//Error
IF timDissableFunctions.Q THEN 
	fbBattery.bWarning := TRUE; 
	fbBattery.iWarningCode := 0; 
ELSE 
	fbBattery.bWarning := FALSE; 
END_IF 
IF (stDataPixii.bError AND stDataPixii.eBatteryState = E_Pixii_BatteryState.eFault) OR timErrorMTCP.Q OR Lynus_Standards.GVL_Energy.stNumberOfDevices.diNumberOfBatterys > Constants_Energy.diMaxNumberOfBatterys THEN 
	fbBattery.bError := TRUE; 
ELSE 
	fbBattery.bError := FALSE; 
END_IF
IF Lynus_Standards.GVL_Energy.stNumberOfDevices.diNumberOfBatterys > Constants_Energy.diMaxNumberOfBatterys THEN 
	fbBattery.iErrorCode := 1;
ELSIF stDataPixii.bError THEN 
	fbBattery.iErrorCode := 0; 
END_IF

//Function
fbBattery(
	bEnable:= bEnable AND NOT timDissableFunctions.Q, 
	bError:= , 
	bWarning:= , 
	bCalculatePower:= TRUE, 
	bReset:= bReset OR timReset.Q, 
	bWriteWithDelay:= TRUE, 
	iErrorCode:= , 
	iWarningCode:= , 
	dwBatterySOC:= , 
	dwBatterySOH:= 0, 
	rBatteryVoltage:= , 
	rMaxDcChargeCurrentBattery:= , 
	rMaxDcDischargeCurrentBattery:= , 
	rMaxChargeVoltage:= 0, 
	lrMaxCapacityBattery:= lrMaxCapacityBattery, 
	lrBatteryPower:= 0, 
	lrBatteryCurrent:= , 
	lrBatteryTemp:= , 
	tTimDelayOutput:= T#5S, 
	stDataBatteryOut=> , 
	stDataBatteryOutDelay=> stDataBatt);


(*------------------------------------------------------------------------------------------State Machine Write---------------------------------------------------------------------------------------------*)	
	
CASE iStateModbusWrite OF	
	
	1://Setpoint for Power 
		iStateModbus_CP := iStateModbusWrite;	
		
		//fbMBWrite_FC6.nQuantity := 2;
		fbMBWrite_FC6.nMBAddr := 39904;
		fbMBWrite_FC6.bExecute := TRUE;
	
		//Setpoint for the Power when discharge (in kW on the Inverter) 
		IF fbBatteryInverter.stDataBattInvertOut.rTargetPower >= 0 THEN
			IF 	((fbBatteryInverter.stDataBattInvertOut.rMaxDischargePower /100) * (fbBatteryInverter.stDataBattInvertOut.rTargetPower * 100)) >= - 32768 AND 
				((fbBatteryInverter.stDataBattInvertOut.rMaxDischargePower /100) * (fbBatteryInverter.stDataBattInvertOut.rTargetPower * 100)) <= 32767 THEN
					iSetpointPower := REAL_TO_INT((fbBatteryInverter.stDataBattInvertOut.rMaxDischargePower / 100) * (fbBatteryInverter.stDataBattInvertOut.rTargetPower * 100));  
					wordBuffer_FC6 := INT_TO_WORD(iSetpointPower);
			END_IF
		END_IF
		//Setpoint for the Power when charge (in kW on the Inverter) 
		IF fbBatteryInverter.stDataBattInvertOut.rTargetPower < 0 OR fbPIDChrgStandby.bEnable THEN
			IF 	((fbBatteryInverter.stDataBattInvertOut.rMaxChargePower / 100) * (fbBatteryInverter.stDataBattInvertOut.rTargetPower * 100)) >= - 32768 AND 
				((fbBatteryInverter.stDataBattInvertOut.rMaxChargePower / 100) * (fbBatteryInverter.stDataBattInvertOut.rTargetPower * 100)) <= 32767 THEN
					iSetpointPower := REAL_TO_INT((fbBatteryInverter.stDataBattInvertOut.rMaxChargePower / 100) * (fbBatteryInverter.stDataBattInvertOut.rTargetPower * 100));  
					//Take the Setpoint from the Standby Controller
					IF fbPIDChrgStandby.bEnable AND fbPIDChrgStandby.rQController <= 0 AND fbPIDChrgStandby.rQController >= -32768 THEN
						iSetpointPower := REAL_TO_INT(fbPIDChrgStandby.rQController);  
					END_IF
					wordBuffer_FC6 := INT_TO_WORD(iSetpointPower); 
			END_IF
		END_IF
		//manual operation setpoint, for testing pupose only!
		IF m_ManualSetpointEnable THEN
			wordBuffer_FC6 := INT_TO_WORD(i_SetpointPower_Manual_kW*10); 
		END_IF
		iSetpointPower_Info := WORD_TO_INT(WordBuffer_FC6);
		
		IF fbMBWrite_FC6.bBusy THEN 
			timDelay.IN := TRUE; 
		END_IF

		//Wait for Delay and then next step
		IF NOT fbMBWrite_FC6.bBusy AND NOT fbMBWrite_FC6.bError AND timDelay.Q THEN
			fbMBWrite_FC6.bExecute := FALSE;
			timDelay.IN := FALSE;
			stDataPixii.bError := FALSE; 
			stDataPixii.eErrorState := E_Pixii_Error.eNormal;
			//Restart from new with the Read out part
			iStateModbusRead := 0;
			iStateModbusWrite := 10;
		END_IF
				
		//Error or Timout
		IF FPError_FC_6.Q OR timTimeout.Q THEN
			iStateModbusError := 300;
			stDataPixii.eErrorState := E_Pixii_Error.eModbusTCPError;
		END_IF

	10:// waite one cycle and count handshake counter +1
		int_Handshake_Counter := int_Handshake_Counter+1;
		iStateModbusWrite := 11;
	
	11:// write handshake timeout +1
		iStateModbus_CP := iStateModbusWrite;	
		
		//fbMBWrite_FC6.nQuantity := 2;
		fbMBWrite_FC6.nMBAddr := 39903;
		fbMBWrite_FC6.bExecute := TRUE;
	
		wordBuffer_FC6 := INT_TO_WORD(int_Handshake_Counter); 
		
		IF fbMBWrite_FC6.bBusy THEN 
			timDelay.IN := TRUE; 
		END_IF

		//Wait for Delay and then next step
		IF NOT fbMBWrite_FC6.bBusy AND NOT fbMBWrite_FC6.bError AND timDelay.Q THEN
			fbMBWrite_FC6.bExecute := FALSE;
			timDelay.IN := FALSE;
			stDataPixii.bError := FALSE; 
			stDataPixii.eErrorState := E_Pixii_Error.eNormal;
			//Restart from new with the Read out part
			iStateModbusRead := 1;
			iStateModbusWrite := 0;
		END_IF
				
		//Error or Timout
		IF FPError_FC_6.Q OR timTimeout.Q THEN
			iStateModbusError := 300;
			stDataPixii.eErrorState := E_Pixii_Error.eModbusTCPError;
		END_IF

END_CASE

(*------------------------------------------------------------------------------------------State Machine Write---------------------------------------------------------------------------------------------*)	

CASE iStateModbusError OF
	
	300://Error
		iStateModbus_CP := iStateModbusError;
		timDelay.IN := FALSE;
		fbMBRead_FC3.bExecute := FALSE;
		fbMBWrite_FC6.bExecute := FALSE;
		stDataPixii.bError := TRUE;	
		//Restart from new with the Read out part after an Error
		iStateModbusRead := 1;	
		iStateModbusError := 0;
		iStateModbusWrite := 0;
END_CASE

(*------------------------------------------------------------------------------------------Modbus TCP Functions---------------------------------------------------------------------------------------------*)

fbMBRead_FC3(	sIPAddr:= sIPAdress, 
				nUnitID := byUnitID, 
				nTCPPort:= 502, 
				cbLength:= SIZEOF(arrBuffer_FC3), 
				pDestAddr:= ADR(arrBuffer_FC3), 
				tTimeout:= T#10S );
FPError_FC_3(	CLK:= fbMBRead_FC3.bError, 
				Q=> );

fbMBWrite_FC6(	sIPAddr:= sIPAdress, 
				nTCPPort:= 502, 
				nUnitID:= byUnitID, 
				nMBAddr:= , 
				nValue:= wordBuffer_FC6, 
				bExecute:= , 
				tTimeout:=  T#10S, 
				bBusy=> , 
				bError=> , 
				nErrId=> );				

FPError_FC_6(	CLK:= fbMBWrite_FC6.bError, 
				Q=> );


				
//Function
fbEMPower(
	bEnable:= bEnable AND NOT timDissableFunctions.Q, 
	bError:= , 
	bEnableReadOutFunction:= FALSE, 
	bWriteWithDelay:= TRUE, 
	bPowerDataInvers:= FALSE,
	bReadOutDataDone:= ,
	iTimeReadOutInterval:= , 
	iErrorCode:= , 
	iWarningCode:= , 
	lrTotalCounterEnergy_Consumption:= , 
	lrTotalCounterEnergy_Production:= , 
	lrCounterEnergyT1_Consumption:= , 
	lrCounterEnergyT2_Consumption:= 0, 
	lrCounterEnergyT1_Production:= , 
	lrCounterEnergyT2_Production:= 0, 
	lrCurrentL1:= , 
	lrVoltageL1N:= , 
	lrVoltageL1L2:= , 
	lrPowerL1:= 0, 
	lrCurrentL2:= , 
	lrVoltageL2N:= , 
	lrVoltageL2L3:= , 
	lrPowerL2:= 0, 
	lrCurrentL3:= , 
	lrVoltageL3N:= , 
	lrVoltageL3L1:= , 
	lrPowerL3:= 0, 
	lrPowerTotal:= , 
	lrFrequency:= , 
	lrReactivePowerTotal:= , 
	lrApparentPowerTotal:= 0, 
	tTimDelayOutput:= T#5S, 
	stDataEMOutPower=> , 
	stDataEMOutPowerDelay=> stDataEMPower, 
	stDataEMOutCounter=> ,
	stDataEMOutCounterDelay=> stDataEMCounter,  
	bReadOutMeter=> );
(*-----------------------------------------------------------Handle data to Global structure for al Devices that are included in this function-----------------------------------------------------------------*)

//Delete al old Data on GVL after a online change or change on the variable diNrOfEMS_IDOD
IF diNrOfEMS_IN <> diNrOfEMS_IN_CP AND iStateGVLData = 0 THEN 
	iStateGVLData := 10; 
END_IF 

CASE iStateGVLData OF
	
	0://Init Step
		byWaitInStep := 0;
		arrCounterForGVL[1] := 1; arrCounterForGVL[2] := 1; arrCounterForGVL[3] := 1;
	
	1://Wait for 4 Steps before clean al Data on GVL
		byWaitInStep := byWaitInStep + 1;
		IF (byWaitInStep >= 4 AND (fbNumberDeviceBattery.bNumberIsCalculatet OR fbNumberDeviceBatteryInvert.bNumberIsCalculatet OR fbNumberDeviceGrid.bNumberIsCalculatet)) THEN 
			iStateGVLData := 2; 
		END_IF
		//To much Devices, back to the Init step
		IF byWaitInStep >= 4 AND NOT fbNumberDeviceBattery.bNumberIsCalculatet AND NOT fbNumberDeviceBatteryInvert.bNumberIsCalculatet AND NOT fbNumberDeviceGrid.bNumberIsCalculatet THEN 
			iStateGVLData := 0; 
		END_IF	
			
	2://Clear all Data in GVL
		FOR diLPForGVL := 1 TO Constants_Energy.diMaxNumberOfEMS BY 1 DO
			//Battery Inverters 
			IF fbNumberDeviceBatteryInvert.bNumberIsCalculatet THEN 
				Lynus_Standards.GVL_Energy.stDataOfBatteryInverters[diLPForGVL,arrCounterForGVL[1]].bEnabled := FALSE;
				Lynus_Standards.GVL_Energy.stDataOfBatteryInverters[diLPForGVL,arrCounterForGVL[1]].bOnOff := FALSE;
				Lynus_Standards.GVL_Energy.stDataOfBatteryInverters[diLPForGVL,arrCounterForGVL[1]].bWorkOnIslandMode := FALSE;
				Lynus_Standards.GVL_Energy.stDataOfBatteryInverters[diLPForGVL,arrCounterForGVL[1]].byErrorWarning := 0;
				Lynus_Standards.GVL_Energy.stDataOfBatteryInverters[diLPForGVL,arrCounterForGVL[1]].byPriority := 0;
				Lynus_Standards.GVL_Energy.stDataOfBatteryInverters[diLPForGVL,arrCounterForGVL[1]].dwBatterySOC := 0;
				Lynus_Standards.GVL_Energy.stDataOfBatteryInverters[diLPForGVL,arrCounterForGVL[1]].lrPowerOnIslandMode := 0;
				Lynus_Standards.GVL_Energy.stDataOfBatteryInverters[diLPForGVL,arrCounterForGVL[1]].rMaxChargePower := 0;
				Lynus_Standards.GVL_Energy.stDataOfBatteryInverters[diLPForGVL,arrCounterForGVL[1]].rMaxDischargePower := 0;
				Lynus_Standards.GVL_Energy.stDataOfBatteryInverters[diLPForGVL,arrCounterForGVL[1]].lrPowerNormalMode := 0;
				//Set also the target value from ems back here to 0 and not in EMS function because EMS is in Standy when we have a online change (Problem when we delete a ems function and make a online change)
				Lynus_Standards.GVL_Energy.stDataOfBatteryInverters[diLPForGVL,arrCounterForGVL[1]].rTargetPowerEMS := 0;
				Lynus_Standards.GVL_Energy.stDataOfBatteryInverters[diLPForGVL,arrCounterForGVL[1]].byMaxDepthOfDischargeEPO := 0;
				Lynus_Standards.GVL_Energy.stDataOfBatteryInverters[diLPForGVL,arrCounterForGVL[1]].byReserveSOCEPO := 0;
			END_IF
			//Batterys 
			IF fbNumberDeviceBattery.bNumberIsCalculatet THEN 
				Lynus_Standards.GVL_Energy.stDataOfBatterys[diLPForGVL,arrCounterForGVL[2]].bEnabled := FALSE;
				Lynus_Standards.GVL_Energy.stDataOfBatterys[diLPForGVL,arrCounterForGVL[2]].byErrorWarning := 0;
				Lynus_Standards.GVL_Energy.stDataOfBatterys[diLPForGVL,arrCounterForGVL[2]].dwSOC := 0;
				Lynus_Standards.GVL_Energy.stDataOfBatterys[diLPForGVL,arrCounterForGVL[2]].dwSOH := 0;
				Lynus_Standards.GVL_Energy.stDataOfBatterys[diLPForGVL,arrCounterForGVL[2]].lrCapacity := 0;
				Lynus_Standards.GVL_Energy.stDataOfBatterys[diLPForGVL,arrCounterForGVL[2]].lrCurrent := 0;
				Lynus_Standards.GVL_Energy.stDataOfBatterys[diLPForGVL,arrCounterForGVL[2]].lrPower := 0;
				Lynus_Standards.GVL_Energy.stDataOfBatterys[diLPForGVL,arrCounterForGVL[2]].lrPowerConsumption := 0;
				Lynus_Standards.GVL_Energy.stDataOfBatterys[diLPForGVL,arrCounterForGVL[2]].lrPowerProduction := 0;
				Lynus_Standards.GVL_Energy.stDataOfBatterys[diLPForGVL,arrCounterForGVL[2]].lrTemp := 0;
				Lynus_Standards.GVL_Energy.stDataOfBatterys[diLPForGVL,arrCounterForGVL[2]].rMaxChargeVoltage := 0;
				Lynus_Standards.GVL_Energy.stDataOfBatterys[diLPForGVL,arrCounterForGVL[2]].rMaxDcChargeCurrent := 0;
				Lynus_Standards.GVL_Energy.stDataOfBatterys[diLPForGVL,arrCounterForGVL[2]].rMaxDcDischargeCurrent := 0;
				Lynus_Standards.GVL_Energy.stDataOfBatterys[diLPForGVL,arrCounterForGVL[2]].rVoltage := 0;
			END_IF
		END_FOR
		//Electric Meter Grid
		IF fbNumberDeviceGrid.bNumberIsCalculatet THEN 
			Lynus_Standards.GVL_Energy.stDataElectricMeters[arrCounterForGVL[3]].bEnabled := FALSE;	
			Lynus_Standards.GVL_Energy.stDataElectricMeters[arrCounterForGVL[3]].byErrorWarning := 0;
			Lynus_Standards.GVL_Energy.stDataElectricMeters[arrCounterForGVL[3]].lrCounterEnergyT1_Consumption := 0;
			Lynus_Standards.GVL_Energy.stDataElectricMeters[arrCounterForGVL[3]].lrCounterEnergyT1_Production := 0;
			Lynus_Standards.GVL_Energy.stDataElectricMeters[arrCounterForGVL[3]].lrCounterEnergyT2_Consumption := 0;
			Lynus_Standards.GVL_Energy.stDataElectricMeters[arrCounterForGVL[3]].lrCounterEnergyT2_Production := 0;
			Lynus_Standards.GVL_Energy.stDataElectricMeters[arrCounterForGVL[3]].lrPower := 0;
			Lynus_Standards.GVL_Energy.stDataElectricMeters[arrCounterForGVL[3]].lrPowerConsumption := 0;
			Lynus_Standards.GVL_Energy.stDataElectricMeters[arrCounterForGVL[3]].lrPowerProduction := 0;
			Lynus_Standards.GVL_Energy.stDataElectricMeters[arrCounterForGVL[3]].lrTotalCounterEnergy_Consumption := 0;
			Lynus_Standards.GVL_Energy.stDataElectricMeters[arrCounterForGVL[3]].lrTotalCounterEnergy_Production := 0;
		END_IF
		
		//Counter for Battery Inverter
		arrCounterForGVL[1] := arrCounterForGVL[1] + 1;
		arrCounterForGVL[1] := LIMIT(0,arrCounterForGVL[1],Constants_Energy.diMaxNumberOfBatteryInverters);
		//Counter for Batterys
		arrCounterForGVL[2] := arrCounterForGVL[2] + 1;
		arrCounterForGVL[2] := LIMIT(0,arrCounterForGVL[2],Constants_Energy.diMaxNumberOfBatterys);
		//Electric Meters
		arrCounterForGVL[3] := arrCounterForGVL[3] + 1;
		arrCounterForGVL[3] := LIMIT(0,arrCounterForGVL[3],Constants_Energy.diMaxNumberOfElectricMeters);
		//Back to the init step
		IF arrCounterForGVL[1] >= Constants_Energy.diMaxNumberOfBatteryInverters AND arrCounterForGVL[2] >= Constants_Energy.diMaxNumberOfBatterys AND arrCounterForGVL[3] >= Constants_Energy.diMaxNumberOfElectricMeters THEN 
			iStateGVLData := 0; 
		END_IF

	10://Clear old Data on GVL 		
		//Battery Inverter
		Lynus_Standards.GVL_Energy.stDataOfBatteryInverters[diNrOfEMS_IN_CP,diNrOfBattInverter_OUT].bEnabled := FALSE;
		Lynus_Standards.GVL_Energy.stDataOfBatteryInverters[diNrOfEMS_IN_CP,diNrOfBattInverter_OUT].bOnOff := FALSE;
		Lynus_Standards.GVL_Energy.stDataOfBatteryInverters[diNrOfEMS_IN_CP,diNrOfBattInverter_OUT].bWorkOnIslandMode := FALSE;
		Lynus_Standards.GVL_Energy.stDataOfBatteryInverters[diNrOfEMS_IN_CP,diNrOfBattInverter_OUT].byErrorWarning := 0;
		Lynus_Standards.GVL_Energy.stDataOfBatteryInverters[diNrOfEMS_IN_CP,diNrOfBattInverter_OUT].byPriority := 0;
		Lynus_Standards.GVL_Energy.stDataOfBatteryInverters[diNrOfEMS_IN_CP,diNrOfBattInverter_OUT].dwBatterySOC := 0;
		Lynus_Standards.GVL_Energy.stDataOfBatteryInverters[diNrOfEMS_IN_CP,diNrOfBattInverter_OUT].lrPowerOnIslandMode := 0;
		Lynus_Standards.GVL_Energy.stDataOfBatteryInverters[diNrOfEMS_IN_CP,diNrOfBattInverter_OUT].rMaxChargePower := 0;
		Lynus_Standards.GVL_Energy.stDataOfBatteryInverters[diNrOfEMS_IN_CP,diNrOfBattInverter_OUT].rMaxDischargePower := 0;
		Lynus_Standards.GVL_Energy.stDataOfBatteryInverters[diNrOfEMS_IN_CP,diNrOfBattInverter_OUT].lrPowerNormalMode := 0;
		//Batterys		
		Lynus_Standards.GVL_Energy.stDataOfBatterys[diNrOfEMS_IN_CP,diNrOfBatt_OUT].bEnabled := FALSE;
		Lynus_Standards.GVL_Energy.stDataOfBatterys[diNrOfEMS_IN_CP,diNrOfBatt_OUT].byErrorWarning := 0;
		Lynus_Standards.GVL_Energy.stDataOfBatterys[diNrOfEMS_IN_CP,diNrOfBatt_OUT].dwSOC := 0;
		Lynus_Standards.GVL_Energy.stDataOfBatterys[diNrOfEMS_IN_CP,diNrOfBatt_OUT].dwSOH := 0;
		Lynus_Standards.GVL_Energy.stDataOfBatterys[diNrOfEMS_IN_CP,diNrOfBatt_OUT].lrCapacity := 0;
		Lynus_Standards.GVL_Energy.stDataOfBatterys[diNrOfEMS_IN_CP,diNrOfBatt_OUT].lrCurrent := 0;
		Lynus_Standards.GVL_Energy.stDataOfBatterys[diNrOfEMS_IN_CP,diNrOfBatt_OUT].lrPower := 0;
		Lynus_Standards.GVL_Energy.stDataOfBatterys[diNrOfEMS_IN_CP,diNrOfBatt_OUT].lrPowerConsumption := 0;
		Lynus_Standards.GVL_Energy.stDataOfBatterys[diNrOfEMS_IN_CP,diNrOfBatt_OUT].lrPowerProduction := 0;
		Lynus_Standards.GVL_Energy.stDataOfBatterys[diNrOfEMS_IN_CP,diNrOfBatt_OUT].lrTemp := 0;
		Lynus_Standards.GVL_Energy.stDataOfBatterys[diNrOfEMS_IN_CP,diNrOfBatt_OUT].rMaxChargeVoltage := 0;
		Lynus_Standards.GVL_Energy.stDataOfBatterys[diNrOfEMS_IN_CP,diNrOfBatt_OUT].rMaxDcChargeCurrent := 0;
		Lynus_Standards.GVL_Energy.stDataOfBatterys[diNrOfEMS_IN_CP,diNrOfBatt_OUT].rMaxDcDischargeCurrent := 0;
		Lynus_Standards.GVL_Energy.stDataOfBatterys[diNrOfEMS_IN_CP,diNrOfBatt_OUT].rVoltage := 0;
									
		diNrOfEMS_IN_CP := diNrOfEMS_IN;
		//Back to the init step
		iStateGVLData := 0;

END_CASE 	 

//Write Data on GVL for Battery Inverter
IF diNrOfBattInverter_OUT > 0 AND fbNumberDeviceBatteryInvert.bNumberIsCalculatet AND diNrOfEMS_IN > 0 THEN
	Lynus_Standards.GVL_Energy.stDataOfBatteryInverters[diNrOfEMS_IN,diNrOfBattInverter_OUT].bEnabled := fbBatteryInverter.stDataBattInvertOut.bEnabled;
	Lynus_Standards.GVL_Energy.stDataOfBatteryInverters[diNrOfEMS_IN,diNrOfBattInverter_OUT].bOnOff := fbBatteryInverter.stDataBattInvertOut.bOnOff;
	Lynus_Standards.GVL_Energy.stDataOfBatteryInverters[diNrOfEMS_IN,diNrOfBattInverter_OUT].bWorkOnIslandMode := fbBatteryInverter.stDataBattInvertOut.bWorkOnIslandMode;
	Lynus_Standards.GVL_Energy.stDataOfBatteryInverters[diNrOfEMS_IN,diNrOfBattInverter_OUT].byErrorWarning := fbBatteryInverter.stDataBattInvertOut.byErrorWarning;
	Lynus_Standards.GVL_Energy.stDataOfBatteryInverters[diNrOfEMS_IN,diNrOfBattInverter_OUT].byPriority := fbBatteryInverter.stDataBattInvertOut.byPriority;
	Lynus_Standards.GVL_Energy.stDataOfBatteryInverters[diNrOfEMS_IN,diNrOfBattInverter_OUT].dwBatterySOC := fbBatteryInverter.dwBatterSOC;
	Lynus_Standards.GVL_Energy.stDataOfBatteryInverters[diNrOfEMS_IN,diNrOfBattInverter_OUT].lrPowerOnIslandMode := fbBatteryInverter.stDataBattInvertOut.lrPowerOnIslandMode;	
	Lynus_Standards.GVL_Energy.stDataOfBatteryInverters[diNrOfEMS_IN,diNrOfBattInverter_OUT].rMaxChargePower := fbBatteryInverter.stDataBattInvertOut.rMaxChargePower;
	Lynus_Standards.GVL_Energy.stDataOfBatteryInverters[diNrOfEMS_IN,diNrOfBattInverter_OUT].rMaxDischargePower := fbBatteryInverter.stDataBattInvertOut.rMaxDischargePower;
	Lynus_Standards.GVL_Energy.stDataOfBatteryInverters[diNrOfEMS_IN,diNrOfBattInverter_OUT].lrPowerNormalMode := fbBatteryInverter.stDataBattInvertOut.lrPowerNormalMode;	
END_IF 
//Write Data on GVL for Batterys
IF diNrOfBatt_OUT > 0 AND fbNumberDeviceBattery.bNumberIsCalculatet AND diNrOfEMS_IN > 0 THEN
	Lynus_Standards.GVL_Energy.stDataOfBatterys[diNrOfEMS_IN,diNrOfBatt_OUT].bEnabled := fbBattery.stDataBatteryOut.bEnabled;	
	Lynus_Standards.GVL_Energy.stDataOfBatterys[diNrOfEMS_IN,diNrOfBatt_OUT].byErrorWarning := fbBattery.stDataBatteryOut.byErrorWarning;
	Lynus_Standards.GVL_Energy.stDataOfBatterys[diNrOfEMS_IN,diNrOfBatt_OUT].dwSOC := fbBattery.stDataBatteryOut.dwSOC;
	Lynus_Standards.GVL_Energy.stDataOfBatterys[diNrOfEMS_IN,diNrOfBatt_OUT].dwSOH := fbBattery.stDataBatteryOut.dwSOH;
	Lynus_Standards.GVL_Energy.stDataOfBatterys[diNrOfEMS_IN,diNrOfBatt_OUT].lrCapacity := fbBattery.stDataBatteryOut.lrCapacity;
	Lynus_Standards.GVL_Energy.stDataOfBatterys[diNrOfEMS_IN,diNrOfBatt_OUT].lrCurrent := fbBattery.stDataBatteryOut.lrCurrent;
	Lynus_Standards.GVL_Energy.stDataOfBatterys[diNrOfEMS_IN,diNrOfBatt_OUT].lrPower := fbBattery.stDataBatteryOut.lrPower;
	Lynus_Standards.GVL_Energy.stDataOfBatterys[diNrOfEMS_IN,diNrOfBatt_OUT].lrPowerConsumption := fbBattery.stDataBatteryOut.lrPowerConsumption;
	Lynus_Standards.GVL_Energy.stDataOfBatterys[diNrOfEMS_IN,diNrOfBatt_OUT].lrPowerProduction := fbBattery.stDataBatteryOut.lrPowerProduction;
	Lynus_Standards.GVL_Energy.stDataOfBatterys[diNrOfEMS_IN,diNrOfBatt_OUT].lrTemp := fbBattery.stDataBatteryOut.lrTemp;
	Lynus_Standards.GVL_Energy.stDataOfBatterys[diNrOfEMS_IN,diNrOfBatt_OUT].rMaxChargeVoltage := fbBattery.stDataBatteryOut.rMaxChargeVoltage;
	Lynus_Standards.GVL_Energy.stDataOfBatterys[diNrOfEMS_IN,diNrOfBatt_OUT].rMaxDcChargeCurrent := fbBattery.stDataBatteryOut.rMaxDcChargeCurrent;
	Lynus_Standards.GVL_Energy.stDataOfBatterys[diNrOfEMS_IN,diNrOfBatt_OUT].rMaxDcDischargeCurrent := fbBattery.stDataBatteryOut.rMaxDcDischargeCurrent;
	Lynus_Standards.GVL_Energy.stDataOfBatterys[diNrOfEMS_IN,diNrOfBatt_OUT].rVoltage := fbBattery.stDataBatteryOut.rBatteryVoltage;
END_IF
(*
//Write Data on GVL for Electric Meter (Grid)
IF diNrOfEM_OUT_Grid > 0 AND fbNumberDeviceGrid.bNumberIsCalculatet THEN
	Lynus_Standards.GVL_Energy.stDataElectricMeters[diNrOfEM_OUT_Grid].bEnabled := fbEMGrid.stDataEMOutPower.bEnabled;
	Lynus_Standards.GVL_Energy.stDataElectricMeters[diNrOfEM_OUT_Grid].byErrorWarning := fbEMGrid.stDataEMOutPower.byErrorWarning;
	Lynus_Standards.GVL_Energy.stDataElectricMeters[diNrOfEM_OUT_Grid].lrCounterEnergyT1_Consumption := fbEMGrid.stDataEMOutCounter.lrCounterEnergyT1_Consumption;
	Lynus_Standards.GVL_Energy.stDataElectricMeters[diNrOfEM_OUT_Grid].lrCounterEnergyT1_Production := fbEMGrid.stDataEMOutCounter.lrCounterEnergyT1_Production;
	Lynus_Standards.GVL_Energy.stDataElectricMeters[diNrOfEM_OUT_Grid].lrCounterEnergyT2_Consumption := fbEMGrid.stDataEMOutCounter.lrCounterEnergyT2_Consumption;
	Lynus_Standards.GVL_Energy.stDataElectricMeters[diNrOfEM_OUT_Grid].lrCounterEnergyT2_Production := fbEMGrid.stDataEMOutCounter.lrCounterEnergyT2_Production;		
	Lynus_Standards.GVL_Energy.stDataElectricMeters[diNrOfEM_OUT_Grid].lrPower := fbEMGrid.stDataEMOutPower.lrPowerTotal;
	Lynus_Standards.GVL_Energy.stDataElectricMeters[diNrOfEM_OUT_Grid].lrPowerConsumption := fbEMGrid.stDataEMOutPower.lrPowerConsumption;
	Lynus_Standards.GVL_Energy.stDataElectricMeters[diNrOfEM_OUT_Grid].lrPowerProduction := fbEMGrid.stDataEMOutPower.lrPowerProduction;
	Lynus_Standards.GVL_Energy.stDataElectricMeters[diNrOfEM_OUT_Grid].lrTotalCounterEnergy_Consumption := fbEMGrid.stDataEMOutCounter.lrTotalCounterEnergy_Consumption;
	Lynus_Standards.GVL_Energy.stDataElectricMeters[diNrOfEM_OUT_Grid].lrTotalCounterEnergy_Production := fbEMGrid.stDataEMOutCounter.lrTotalCounterEnergy_Production;
END_IF
*)
(*----------------------------------------------------------Save persistent data----------------------------------------------------------------*)

arrPD[1](lrValue:= BOOL_TO_LREAL(bEnable), bEventBasedActive=> );
arrPD[2](lrValue:= BOOL_TO_LREAL(bActivateControl), bEventBasedActive=> );
arrPD[3](lrValue:= BYTE_TO_LREAL(byUnitID), bEventBasedActive=> );
arrPD[4](lrValue:= BYTE_TO_LREAL(byPriority), bEventBasedActive=> );
arrPD[5](lrValue:= DINT_TO_LREAL(diNrOfEMS_IN), bEventBasedActive=> );
arrPD[6](lrValue:= lrMaxCapacityBattery, bEventBasedActive=> );
arrPD[7](lrValue:= DINT_TO_LREAL(diNrOfEMS_IN_CP), bEventBasedActive=> );
PD_String(sText:= sIPAdress, bEventBasedActive=> );

END_FUNCTION_BLOCK

// ---- FBs/Schneider/FB_Schneider_EVlinkWallbox.TcPOU
FUNCTION_BLOCK FB_Schneider_EVlinkWallbox
VAR_INPUT PERSISTENT
	bEnable										: BOOL;																			// Enable the Fuctionblock and his logic
	bEnableWrite								: BOOL;																			// Enable Write function 
	bPowerDataInvers							: BOOL;																			//With True its possible to invert all received power data from the electric meter
	byElectricFuseLine							: BYTE; 																		//Electric Fuse Line on wich the ECS is connected => 1 2 3 (If 0 then this charging station is not connected to a Electric Fuse Line)
	rMinCurrent									: REAL:=6;																		// min Current e.g. 6A	max 32A	
	diNrOfEMS_IN								: DINT;																			//Number of EMS what control this Device.
	diNrOfEM_IN_CS								: DINT;																			//Number of the electric meter for incoming power data. (Power Data for this Device)
	sIPAdress									: STRING(15);																	//IP Adress from the charging station
	stSetupECS									: ST_Setup_ECS;																	//{#lynus.ag#()} //Setup charging station
END_VAR
VAR_OUTPUT
	stDataECS									: ST_ECS_Output;																//{#lynus.ag#()} //Electric charging station output data
	diNrOfECS_OUT								: DINT;																			//Active Number from the Electric charging Function for using on other functions
	lrTotalPowerECSRealTime						: LREAL;																		//Total Electric Power in kW read out directly from the Charging station. (Real time)
	stDataElectric								: ST_ElectricMeter_Output_Power;												// Electrict data from the charging station
	str_Mode3State								: STRING(2);																	//Mode 3 State
	bErrorCS									: BOOL;																			//Error State from the charging station
	lrTotalCounterEnergy_Consumption			: LREAL;																		//Energy Counter Consumption in Wh
	bCarConnected								: BOOL;																			// Car Connected

END_VAR
VAR
	{attribute 'hide'}
	fbCS										: FB_ElectricChargingStation;													//Function block for electric charging station
	{attribute 'hide'}
	fbNumberDevice								: FB_NumberOfDevice;															//Function block to calcualte the number of the Device
	{attribute 'hide'}
	fbMBRead_FC3								: FB_MBReadRegs;																//Modbus Read Function (FC3)
	{attribute 'hide'}
	fbMBWrite_FC16								: FB_MBWriteRegs;																//Modbus Write Function (FC16)
	{attribute 'hide'}
	fbConvertWordToByte							: FB_CV_WORD_TO_BYTE;															//Convert Word To Byte
	{attribute 'hide'}
	fbConvertDwordToWord						: FB_CV_DWORD_TO_WORD;															//Convert Dword to Word
	{attribute 'hide'}
	fbConvertWordToDword						: FB_CV_WORD_TO_DWORD;															//Convert Word to Dword
	{attribute 'hide'}
	fbConvertWordToUlint						: FB_CV_WORD_TO_ULINT;															//Convert Word to ULINT
	{attribute 'hide'}
	timDelay									: TON;																			//Timer for Delay between Requests
	{attribute 'hide'}
	timTimeout									: TON;																			//Timer for Timeout
	{attribute 'hide'}
	timDissableFunctions						: TON;																			//Timer to dissable the Function after Lynus_Standards.Constants_General.tTimeDissableLynusFunctions Days without connection to the Lynus Cloud
	{attribute 'hide'}
	timResetConnectionOnGVL						: TON;																			//Timer to try reset the connection Flag on the GVL. (When somebody delete the Connection Function and make only a onlinechange)
	{attribute 'hide'}
	timChTimeSocket1							: TON;																			//Charging Time for socket 1
	{attribute 'hide'}
	timChTimeSocket2							: TON;																			//Charging Time for socket 2
	{attribute 'hide'}
	timDelayStart								: TON;																			//Timer to start the state machine with Daley after enabling or after the system ist restartet
	{attribute 'hide'}
	FPError_FC_3								: R_TRIG;																		//Internal positive Edge
	{attribute 'hide'}
	FPError_FC_16								: R_TRIG;																		//Internal positive Edge
	{attribute 'hide'}
	FPEnable									: R_TRIG;																		//Internal positive Edge
	{attribute 'hide'}
	stConvertFloat								: ST_UN_FLOAT_CONVERT_DWORD_REAL;												//Convert float
	{attribute 'hide'}
	stConvertFloat2								: ST_UN_FLOAT_CONVERT_ULINT_LREAL;												//Convert float
	{attribute 'hide'}
	arrPD										: ARRAY[1..18] OF FB_PersistentData_Number;										//Function to save persistent data
	{attribute 'hide'}
	fbPDString									: FB_PersistentData_String;														//Function to save persistent string data
	{attribute 'hide'}
	arrBuffer_FC3								: ARRAY[1..30] OF WORD;															//Buffer with Data from FC3
	{attribute 'hide'}
	arrBuffer_FC16								: ARRAY[1..2] OF WORD;															//Buffer with Data from FC16
	{attribute 'hide'}
	bMBTCPError									: BOOL;																			//Modbus TCP Function Error
	{attribute 'hide'}
	byWaitInStep								: BYTE;																			//Wait in Step before start to clean data on PLC
	{attribute 'hide'}
	iStateGVLData								: INT;																			//State machine to handle the data on the GVL
	{attribute 'hide'}
	iStateModbusRead							: INT;																			//State machine for read out Data over Modbus RTU
	{attribute 'hide'}
	iStateModbusWrite							: INT;																			//State machine for write Data over Modbus RTU
	{attribute 'hide'}
	iStateModbusError							: INT;																			//State machine for error out Data over Modbus RTU	
	{attribute 'hide'}
	iStateModbus_CP								: INT;																			//Variable to compare the state machine variable to set or reset the timeout timer
	{attribute 'hide'}
	diNumberOfActiveBatterys					: DINT;																			//Number of active batterys
	{attribute 'hide'}
	diNumberOfBatteryInverterInEPO				: DINT;																			//Number of battery inverters that work in Emergency Power operation 
	{attribute 'hide'}
	diLPForGVL									: DINT;																			//Loop to clean old data on GVL
	{attribute 'hide'}
	diCounterForGVL								: DINT;																			//Counter to clean old data on GVL
	{attribute 'hide'}
	dwSumSOC									: DWORD;																		//Sum of the SOC from all batterys
	{attribute 'hide'}
	lrTotalCounterEnergy_Production				: LREAL;																		//Energy Counter Production in Wh 
	{attribute 'hide'}
	rPowerECS									: REAL;																			//Power from the ECS in kW 
	iSuccessCounterRead							:ARRAY[1..2] OF INT;
	iSuccessCounterWrite						:ARRAY[1..2] OF INT;
END_VAR
VAR PERSISTENT
	{attribute 'conditionalshow'}
	diNrOfEMS_IN_CP								: DINT;																			//Number of EMS what control this Device to compare with the original
END_VAR

//Creator : Stefan Lackner
//Company : EfficientIO
//Date : 03.03.2023
//Version : 0.0.0.1

//With this Funcition its possible to communicate with a Schneider EVLink Wallbox over Modbus TCP.
//Its possible to controll the charging station over the charg current
//When the Function send 0 Ampere is switched of, then the charging station is blocked and its not possible to charge
//This Function Block supports Charging stations with maximal 1 sockets

//NOTE for diNr.....Designation => 
//_IN = Here Data come in from other Functions or go out to other functions about the GVL
//_OUT = Here Data go out to other functions about the GVL
(*--------------------------------------------------------------------------------------------Limits-------------------------------------------------------------------------------------*)

diNrOfEMS_IN := LIMIT(0,diNrOfEMS_IN,Constants_Energy.diMaxNumberOfEMS);
diNrOfEM_IN_CS := LIMIT(0,diNrOfEM_IN_CS,Constants_Energy.diMaxNumberOfElectricMeters);
byElectricFuseLine := LIMIT(0,byElectricFuseLine,30);
rMinCurrent	:= LIMIT (0,rMinCurrent,32);


(*------------------------------------------------------------------Power Data----------------------------------------------------------------------------*)

IF diNrOfEM_IN_CS <> 0 THEN
	//Energy Session Input data
	fbCS.bCalculateEnergySession := FALSE;
	IF NOT bPowerDataInvers THEN
		//Energy meter input data for cs Function block
		fbCS.lrCounterEnergyT1_Consumption := Lynus_Standards.GVL_Energy.stDataElectricMeters[diNrOfEM_IN_CS].lrCounterEnergyT1_Production * 1000;
		fbCS.lrCounterEnergyT2_Consumption := Lynus_Standards.GVL_Energy.stDataElectricMeters[diNrOfEM_IN_CS].lrCounterEnergyT2_Production * 1000;
		fbCS.lrCounterEnergyT1_Production := Lynus_Standards.GVL_Energy.stDataElectricMeters[diNrOfEM_IN_CS].lrCounterEnergyT1_Consumption * 1000;
		fbCS.lrCounterEnergyT2_Production := Lynus_Standards.GVL_Energy.stDataElectricMeters[diNrOfEM_IN_CS].lrCounterEnergyT1_Consumption * 1000;
		fbCS.lrTotalCounterEnergy_Consumption := Lynus_Standards.GVL_Energy.stDataElectricMeters[diNrOfEM_IN_CS].lrTotalCounterEnergy_Production * 1000;
		fbCS.lrTotalCounterEnergy_Production := Lynus_Standards.GVL_Energy.stDataElectricMeters[diNrOfEM_IN_CS].lrTotalCounterEnergy_Consumption * 1000;
		fbCS.lrTotalPowerECS := (Lynus_Standards.GVL_Energy.stDataElectricMeters[diNrOfEM_IN_CS].lrPower * 1000) * - 1;
	ELSE
		//Energy meter input data for cs Function block
		fbCS.lrCounterEnergyT1_Consumption := Lynus_Standards.GVL_Energy.stDataElectricMeters[diNrOfEM_IN_CS].lrCounterEnergyT1_Consumption * 1000;
		fbCS.lrCounterEnergyT2_Consumption := Lynus_Standards.GVL_Energy.stDataElectricMeters[diNrOfEM_IN_CS].lrCounterEnergyT2_Consumption * 1000;
		fbCS.lrCounterEnergyT1_Production := Lynus_Standards.GVL_Energy.stDataElectricMeters[diNrOfEM_IN_CS].lrCounterEnergyT1_Production * 1000;
		fbCS.lrCounterEnergyT2_Production := Lynus_Standards.GVL_Energy.stDataElectricMeters[diNrOfEM_IN_CS].lrCounterEnergyT2_Production * 1000;
		fbCS.lrTotalCounterEnergy_Consumption := Lynus_Standards.GVL_Energy.stDataElectricMeters[diNrOfEM_IN_CS].lrTotalCounterEnergy_Consumption * 1000;
		fbCS.lrTotalCounterEnergy_Production := Lynus_Standards.GVL_Energy.stDataElectricMeters[diNrOfEM_IN_CS].lrTotalCounterEnergy_Production * 1000;
		fbCS.lrTotalPowerECS := Lynus_Standards.GVL_Energy.stDataElectricMeters[diNrOfEM_IN_CS].lrPower * 1000;
	END_IF
ELSE
	//Energy meter input data for cs Function block
	fbCS.lrCounterEnergyT1_Consumption := lrTotalCounterEnergy_Consumption;
	fbCS.lrCounterEnergyT2_Consumption := 0;
	fbCS.lrCounterEnergyT1_Production := lrTotalCounterEnergy_Production;
	fbCS.lrCounterEnergyT2_Production := 0;
	fbCS.lrTotalCounterEnergy_Consumption := lrTotalCounterEnergy_Consumption;
	fbCS.lrTotalCounterEnergy_Production := lrTotalCounterEnergy_Production;
	fbCS.lrTotalPowerECS := rPowerECS;
	//Energy Session Input data
	fbCS.bCalculateEnergySession := TRUE;
	fbCS.arrSocketPowerECS[1] := rPowerECS;
	fbCS.arrSocketPowerECS[2] := 0;
	fbCS.arrSocketPowerECS[3] := 0;
	fbCS.arrSocketPowerECS[4] := 0;
	fbCS.arrSocketEnergySession[1] := lrTotalCounterEnergy_Consumption;
	fbCS.arrSocketEnergySession[2] := 0;
	fbCS.arrSocketEnergySession[3] := 0;
	fbCS.arrSocketEnergySession[4] := 0;
END_IF			

(*-------------------------------------------------------------Calcualte the number of ECS---------------------------------------------------------------*)

fbNumberDevice(
	diActualNumberOfDevices:= Lynus_Standards.GVL_Energy.stNumberOfDevices.diNumberOfECS, 
	diMaxNumberOfDevices:= Constants_Energy.diMaxNumberOfElectricChargingStations, 
	udiCounterOnlineChange:= TwinCAT_SystemInfoVarList._AppInfo.OnlineChangeCnt, 
	bNumberIsCalculatet=> , 
	bFPNumberIsCalculatet=> , 
	bOnlineChange=> , 
	diNumberForThisDevice=> diNrOfECS_OUT, 
	diNumberOfTotalDevices=> );

//Write new Numer on GVL
IF fbNumberDevice.bFPNumberIsCalculatet THEN
	Lynus_Standards.GVL_Energy.stNumberOfDevices.diNumberOfECS := fbNumberDevice.diNumberOfTotalDevices;	
END_IF 

//Delete old Number on GVL
IF fbNumberDevice.bOnlineChange THEN 
	Lynus_Standards.GVL_Energy.stNumberOfDevices.diNumberOfECS := diNrOfECS_OUT;	
		iStateGVLData := 1;
END_IF

(*-------------------------------------------------------------Service from Backend is ready and check the connection to backen for dissabel/enable Function---------------------------------------------------------------*)

//Try to reset the variable for connection on the GVL. When all is normal then the Lynus Mqtt connection function set this variable to true in the next cycle
//When we have no connection to the backend then after Lynus_Standards.Constants_General.tTimeDissableLynusFunctions days the Function is dissabled with all of his functionalities
timResetConnectionOnGVL(IN:= NOT timResetConnectionOnGVL.Q, PT:= T#1H, Q=> , ET=> );
IF timResetConnectionOnGVL.Q THEN Lynus_Standards.GVL_Communicator.bStateConnectionToEnableFunctions := FALSE; END_IF
IF NOT Lynus_Standards.GVL_Communicator.bStateConnectionToEnableFunctions THEN timDissableFunctions.IN := TRUE; ELSE timDissableFunctions.IN := FALSE; END_IF  
timDissableFunctions(IN:= , PT:= Lynus_Standards.Constants_General.tTimeDissableLynusFunctions, Q=> , ET=> );
			
(*--------------------------------------------------------------------------------------------State Machine Read--------------------------------------------------------------------------------------*)

//Timer for Delay
timDelay(IN:= , PT:= T#350MS, Q=> , ET=> );

//Timer for Timeout in Statemachine
IF (iStateModbusRead > 0 AND iStateModbusRead <= 5 AND iStateModbusRead = iStateModbus_CP) OR
	(iStateModbusWrite > 0 AND iStateModbusWrite <= 2 AND iStateModbusWrite = iStateModbus_CP) 
THEN
	timTimeout.IN := TRUE;
ELSE	
	timTimeout.IN := FALSE;
END_IF
//Timeout Timer is dissabled when the Init Step is aktiv or the function is not enabled
IF (iStateModbusRead = 0 AND iStateModbusWrite = 0) OR NOT bEnable THEN timTimeout.IN := FALSE; END_IF
timTimeout(IN:= , PT:= T#10S, Q=> , ET=> );

//Enable with Delay that not all sockets have to be created at the same time
timDelayStart(IN:= bEnable, PT:= T#20MS * diNrOfECS_OUT, Q=> , ET=> );
FPEnable(CLK:= timDelayStart.Q, Q=> );

IF FPEnable.Q AND iStateModbusRead = 0 AND iStateModbusWrite = 0 THEN iStateModbusRead := 1; END_IF		
		
//Not Enabled
IF NOT bEnable THEN iStateModbusRead := 0; iStateModbusError := 0; iStateModbusWrite := 0; END_IF		
		
CASE iStateModbusRead OF

	0://Init Step 
		iStateModbus_CP := 0;
		timDelay.IN := FALSE;
		fbMBRead_FC3.bExecute := FALSE;
		fbMBWrite_FC16.bExecute := FALSE;
		rPowerECS := 0;	
		str_Mode3State := ''; 
		
	1://Read Out the mode 3 State from the charging station (Register 6)
		iStateModbus_CP := iStateModbusRead;
		
		//Reset Write
		fbMBWrite_FC16.bExecute := FALSE;
		
		//Start Read
		fbMBRead_FC3.nQuantity := 6;
		fbMBRead_FC3.nMBAddr := 1;
		fbMBRead_FC3.bExecute := TRUE;
		IF fbMBRead_FC3.bBusy THEN timDelay.IN := TRUE; END_IF
		
		//Wait for Delay, copy Data and then next step
		IF NOT fbMBRead_FC3.bBusy AND NOT fbMBRead_FC3.bError AND timDelay.Q THEN
			//Mode 3 state
			// fbConvertWordToByte(wInputValue:= arrBuffer_FC3[6], eByteOrderForConvert:= eByteOrder.eBigEndian, byOutputValue_1=> , byOutputValue_2=> );
			CASE arrBuffer_FC3[6] OF   // fbConvertWordToByte.byOutputValue_1
				0:	str_Mode3State:='F';		// 0 – Electric Vehicle Supply Equipment not available - state F
				1:	str_Mode3State:='A';		// 1 - Electric Vehicle Supply Equipment available - state A
				2:	str_Mode3State:='A+';		// 2 - Plug detected - state A+
				3:	str_Mode3State:='??';		// 
				4:	str_Mode3State:='B';		// 4 - EV connected – state B
				5:	str_Mode3State:='C-';		// 5 - EV connected – state C-
				6:	str_Mode3State:='D-';		// 6 - EV connected, ventilation required – state D-
				7:	str_Mode3State:='B+';		// 7 - Electric Vehicle Supply Equipment ready - state B+
				8:	str_Mode3State:='C';		// 8 - EV ready - state C
				9:	str_Mode3State:='C+';		// 9 - Charging EV - state C+
				10:	str_Mode3State:='D';		// 10 - EV ready, ventilation required - state D
				11:	str_Mode3State:='D+';		// 11 - Charging EV, ventilation required - state D+
				12:	str_Mode3State:='St';		// 12 - Stop charging
				13:	str_Mode3State:='Al';		// 13 – Alarm
				14:	str_Mode3State:='E';		// 14 - Shortcut – state E
				15:	str_Mode3State:='Co';		// 15 - Digital Com by Electric Vehicle Supply Equipment state
			END_CASE
			iSuccessCounterRead[iStateModbusRead]:=iSuccessCounterRead[iStateModbusRead]+1;
			//Go to Next Step
			fbMBRead_FC3.bExecute := FALSE;
			timDelay.IN := FALSE;		
			iStateModbusRead := 2;
		END_IF	
	
		//Error or Timeout
		IF FPError_FC_3.Q OR timTimeout.Q THEN
			iStateModbusError := 300;
		END_IF
			
	2://Power Data  (Register 350 - 370)
		iStateModbus_CP := iStateModbusRead;
		
		//Start Read
		fbMBRead_FC3.nQuantity := 24;
		fbMBRead_FC3.nMBAddr := 350;
		fbMBRead_FC3.bExecute := TRUE;
		
		IF fbMBRead_FC3.bBusy THEN timDelay.IN := TRUE; END_IF
			
		//Wait for Delay, copy Data and then next step
		IF NOT fbMBRead_FC3.bBusy AND NOT fbMBRead_FC3.bError AND timDelay.Q THEN
	
			// current phase 1
			fbConvertWordToDword(wInputValue_1:= arrBuffer_FC3[1], wInputValue_2:= arrBuffer_FC3[2], eByteOrderForConvert:= eByteOrder.eBigEndian, dwOutputValue =>);
			stConvertFloat.dwRawValue := fbConvertWordToDword.dwOutputValue;
			stDataElectric.bEnabled:=TRUE;			
			stDataElectric.lrCurrentL1:=REAL_TO_LREAL(stConvertFloat.rValueFloat);
			// current phase 2
			fbConvertWordToDword(wInputValue_1:= arrBuffer_FC3[3], wInputValue_2:= arrBuffer_FC3[4], eByteOrderForConvert:= eByteOrder.eBigEndian, dwOutputValue =>);
			stConvertFloat.dwRawValue := fbConvertWordToDword.dwOutputValue;
			stDataElectric.lrCurrentL2:=REAL_TO_LREAL(stConvertFloat.rValueFloat);
			// current phase 3
			fbConvertWordToDword(wInputValue_1:= arrBuffer_FC3[5], wInputValue_2:= arrBuffer_FC3[6], eByteOrderForConvert:= eByteOrder.eBigEndian, dwOutputValue =>);
			stConvertFloat.dwRawValue := fbConvertWordToDword.dwOutputValue;
			stDataElectric.lrCurrentL3:=REAL_TO_LREAL(stConvertFloat.rValueFloat);
			//energy in Wh
			fbConvertWordToDword(wInputValue_1:= arrBuffer_FC3[7], wInputValue_2:= arrBuffer_FC3[8], eByteOrderForConvert:= eByteOrder.eBigEndian, dwOutputValue =>);
			
			lrTotalCounterEnergy_Consumption := DWORD_TO_LREAL(fbConvertWordToDword.dwOutputValue);
			//Power Data in kW
			fbConvertWordToDword(wInputValue_1:= arrBuffer_FC3[9], wInputValue_2:= arrBuffer_FC3[10], eByteOrderForConvert:= eByteOrder.eBigEndian, dwOutputValue =>);
			stConvertFloat.dwRawValue := fbConvertWordToDword.dwOutputValue;
			rPowerECS := INT_TO_REAL(REAL_TO_INT(stConvertFloat.rValueFloat*10))/10;
			stDataElectric.bEnabled:=TRUE;
			stDataElectric.lrPowerTotal:=REAL_TO_LREAL(rPowerECS);
			// voltage phase 1 - phase 2
			fbConvertWordToDword(wInputValue_1:= arrBuffer_FC3[11], wInputValue_2:= arrBuffer_FC3[12], eByteOrderForConvert:= eByteOrder.eBigEndian, dwOutputValue =>);
			stConvertFloat.dwRawValue := fbConvertWordToDword.dwOutputValue;
			stDataElectric.lrVoltageL1L2:=REAL_TO_LREAL(stConvertFloat.rValueFloat);			
			// voltage phase 2 - phase 3
			fbConvertWordToDword(wInputValue_1:= arrBuffer_FC3[13], wInputValue_2:= arrBuffer_FC3[14], eByteOrderForConvert:= eByteOrder.eBigEndian, dwOutputValue =>);
			stConvertFloat.dwRawValue := fbConvertWordToDword.dwOutputValue;
			stDataElectric.lrVoltageL2L3:=REAL_TO_LREAL(stConvertFloat.rValueFloat);			
			// voltage phase 3 - phase 1
			fbConvertWordToDword(wInputValue_1:= arrBuffer_FC3[15], wInputValue_2:= arrBuffer_FC3[16], eByteOrderForConvert:= eByteOrder.eBigEndian, dwOutputValue =>);
			stConvertFloat.dwRawValue := fbConvertWordToDword.dwOutputValue;
			stDataElectric.lrVoltageL3L1:=REAL_TO_LREAL(stConvertFloat.rValueFloat);			
			// voltage phase 1 - Neutral
			fbConvertWordToDword(wInputValue_1:= arrBuffer_FC3[17], wInputValue_2:= arrBuffer_FC3[18], eByteOrderForConvert:= eByteOrder.eBigEndian, dwOutputValue =>);
			stConvertFloat.dwRawValue := fbConvertWordToDword.dwOutputValue;
			stDataElectric.lrVoltageL1N:=REAL_TO_LREAL(stConvertFloat.rValueFloat);			
			// voltage phase 2 - Neutral
			fbConvertWordToDword(wInputValue_1:= arrBuffer_FC3[19], wInputValue_2:= arrBuffer_FC3[20], eByteOrderForConvert:= eByteOrder.eBigEndian, dwOutputValue =>);
			stConvertFloat.dwRawValue := fbConvertWordToDword.dwOutputValue;
			stDataElectric.lrVoltageL2N:=REAL_TO_LREAL(stConvertFloat.rValueFloat);		
			// voltage phase 3 - Neutral
			fbConvertWordToDword(wInputValue_1:= arrBuffer_FC3[21], wInputValue_2:= arrBuffer_FC3[22], eByteOrderForConvert:= eByteOrder.eBigEndian, dwOutputValue =>);
			stConvertFloat.dwRawValue := fbConvertWordToDword.dwOutputValue;
			stDataElectric.lrVoltageL3N:=REAL_TO_LREAL(stConvertFloat.rValueFloat);					
			
			(*
			350	StationMeter Phase1Current_I1	word
			352	StationMeter Phase2Current_I2	word
			354	StationMeter Phase3Current_I3	word
			356	StationMeter ActiveEnergy	word  [Ws]
			358	StationMeter ActivePowerTotal	word
			360	StationMeter L1_L2 Voltage	word
			362	StationMeter L2_L3 Voltage	word
			364	StationMeter L3_L1 Voltage	word
			366	StationMeter L1_N Voltage	word
			368	StationMeter L2_N Voltage	word
			370	StationMeter L3_N Voltage	word
			*)
	
			iSuccessCounterRead[iStateModbusRead]:=iSuccessCounterRead[iStateModbusRead]+1;
			
			//Go to Next Step
			fbMBRead_FC3.bExecute := FALSE;
			timDelay.IN := FALSE;		
			iStateModbusRead := 5;
		END_IF	
	
		//Error or Timeout
		IF FPError_FC_3.Q OR timTimeout.Q THEN
			iStateModbusError := 300;
		END_IF
			
		
	5://Wait 1 Step to reset the delay counter befor start to write
		iStateModbus_CP := iStateModbusRead;
		IF bEnableWrite THEN 	
			iStateModbusWrite := 1;
			//-1 because 0 is the Init Step for Read
			iStateModbusRead := - 1;
		ELSE
			iStateModbusRead := 1;
			iStateModbusWrite := 0;		
		END_IF
		//Error on Master, changes on Inputs or Timeout
		IF timTimeout.Q THEN 
			iStateModbusError := 300;	 
		END_IF
END_CASE


(*------------------------------------------------------------------Error and Warning----------------------------------------------------------------------------*)	
 
IF str_Mode3State = 'A1' THEN bErrorCS := TRUE; ELSE bErrorCS := FALSE; END_IF  

IF timDissableFunctions.Q THEN fbCS.bWarning := TRUE; fbCS.iWarningCode := 0; ELSE fbCS.bWarning := FALSE; END_IF   
IF Lynus_Standards.GVL_Energy.stNumberOfDevices.diNumberOfECS > Constants_Energy.diMaxNumberOfElectricChargingStations OR bErrorCS OR bMBTCPError THEN 
	fbCS.bError := TRUE;
ELSE 
	fbCS.bError := FALSE;
	fbCS.iErrorCode := 0;
END_IF

IF Lynus_Standards.GVL_Energy.stNumberOfDevices.diNumberOfECS > Constants_Energy.diMaxNumberOfElectricChargingStations THEN fbCS.iErrorCode := 1;
ELSIF bErrorCS OR bMBTCPError THEN fbCS.iErrorCode := 0; END_IF

(*------------------------------------------------------------------Logic----------------------------------------------------------------------------*)


//Car connected to the ECS  
IF  str_Mode3State = 'B' OR str_Mode3State = 'C-' OR str_Mode3State = 'D-' OR str_Mode3State = 'C' OR str_Mode3State = 'C+' OR str_Mode3State = 'D' OR str_Mode3State = 'D+' THEN 
	fbCS.bCarConnected := TRUE; 
	bCarConnected := TRUE;
ELSE 
	fbCS.bCarConnected := FALSE;
	bCarConnected := FALSE; 
END_IF 

//Min Current
fbCS.rMinCurrent := rMinCurrent;

//Charging time
IF str_Mode3State = 'C+' OR str_Mode3State = 'D+' THEN timChTimeSocket1.IN := TRUE; ELSE timChTimeSocket1.IN := FALSE; END_IF


IF timChTimeSocket1.IN THEN fbCS.arrSocketChargingTimeInput[1] := TIME_TO_REAL(timChTimeSocket1.ET) / 60000; END_IF
fbCS.arrSocketChargingTimeInput[2] := 0;
fbCS.arrSocketChargingTimeInput[3] := 0;
fbCS.arrSocketChargingTimeInput[4] := 0;

timChTimeSocket1(IN:= , PT:= T#24H, Q=> , ET=> );


//Mode 3 State
fbCS.arrSocketMode3StateECS[1] := str_Mode3State;
fbCS.arrSocketMode3StateECS[2] := '';
fbCS.arrSocketMode3StateECS[3] := '';
fbCS.arrSocketMode3StateECS[4] := '';

//SOC Car
fbCS.arrSOCCar[1] := 0;
fbCS.arrSOCCar[2] := 0;
fbCS.arrSOCCar[3] := 0;
fbCS.arrSOCCar[4] := 0;

//Functionblock ECS
fbCS(
	bEnable:= bEnable AND NOT timDissableFunctions.Q, 
	bError:= ,
	bWarning := ,
	bEPOIsActive:= , 
	bExternalLock:= , 
	bCarConnected:= , 
	bWriteWithDelay:= TRUE, 
	bCalculateEnergySession:= ,
	iErrorCode:= , 
	iWarningCode:= , 
	arrSocketChargingTimeInput:= ,
	arrSOCCar:= , 
	dwBatterySOC:= 100, 
	lrTotalCounterEnergy_Consumption:= , 
	lrTotalCounterEnergy_Production:= , 
	lrCounterEnergyT1_Consumption:= , 
	lrCounterEnergyT2_Consumption:= , 
	lrCounterEnergyT1_Production:= , 
	lrCounterEnergyT2_Production:= , 
	lrTotalPowerECS:= , 
	arrSocketEnergySession:= ,
	rTargetPower:= Lynus_Standards.GVL_Energy.stDataElectricChargingStations[diNrOfEMS_IN,diNrOfECS_OUT].rTargetPowerEMS, 
	rSupplyVoltage:= 692, 
	rMinCurrent:= , 
	tTimDelayOutput:= T#5S, 
	tDelayError:= T#5S,
	arrSocketMode3StateECS:= ,
	arrSocketPowerECS:= ,
	stSetupECS:= stSetupECS, 
	stDataECSOut=> , 
	stDataECSOutDelay=> stDataECS);

//Real time Power for Output
lrTotalPowerECSRealTime := fbCS.stDataECSOut.lrTotalPower;
	
(*------------------------------------------------------------------------------------------State Machine Write---------------------------------------------------------------------------------------------*)	

CASE iStateModbusWrite OF	

	1://Set the charging current (Reg 301)
		iStateModbus_CP := iStateModbusWrite;
		
		fbMBWrite_FC16.nQuantity := 1;
		fbMBWrite_FC16.nMBAddr := 301;
		fbMBWrite_FC16.bExecute := TRUE;
		
		//Prepear the sending Data. Charging power 0..100%
		IF fbCS.stDataECSOut.rTargetPower >= 0 AND fbCS.stDataECSOut.rTargetPower <= 100 THEN 
			arrBuffer_FC16[1] := REAL_TO_WORD(fbCS.stDataECSOut.rTargetChargeCurrent);	 				
		END_IF
		IF fbMBWrite_FC16.bBusy THEN timDelay.IN := TRUE; END_IF

		//Wait for Delay and then next step
		IF NOT fbMBWrite_FC16.bBusy AND NOT fbMBWrite_FC16.bError AND timDelay.Q THEN
			fbMBWrite_FC16.bExecute := FALSE;
			timDelay.IN := FALSE;
			bMBTCPError := FALSE; 
			iSuccessCounterWrite[iStateModbusWrite]:=iSuccessCounterWrite[iStateModbusWrite]+1;
			iStateModbusWrite := 2;
		END_IF
				
		//Error or Timout
		IF FPError_FC_16.Q OR timTimeout.Q THEN
			iStateModbusError := 300;
		END_IF		
	2:	// write Livebit (1) to register 932	
		iStateModbus_CP := iStateModbusWrite;
		
		fbMBWrite_FC16.nQuantity := 1;
		fbMBWrite_FC16.nMBAddr := 932;
		fbMBWrite_FC16.bExecute := TRUE;
		
		//Prepear the sending Data. Allways write 1 into the regiseter 
		arrBuffer_FC16[1]:=1;
						
		
		IF fbMBWrite_FC16.bBusy THEN timDelay.IN := TRUE; END_IF

		//Wait for Delay and then next step
		IF NOT fbMBWrite_FC16.bBusy AND NOT fbMBWrite_FC16.bError AND timDelay.Q THEN
			fbMBWrite_FC16.bExecute := FALSE;
			timDelay.IN := FALSE;
			bMBTCPError := FALSE; 
			iSuccessCounterWrite[iStateModbusWrite]:=iSuccessCounterWrite[iStateModbusWrite]+1;
			//Restart from new with the Read out part
			iStateModbusRead := 1;
			iStateModbusWrite := 0;
		END_IF
		//Error or Timout
		IF FPError_FC_16.Q OR timTimeout.Q THEN
			iStateModbusError := 300;
		END_IF		
		
END_CASE	
	
(*------------------------------------------------------------------------------------------State Machine Error---------------------------------------------------------------------------------------------*)	

CASE iStateModbusError OF
	
	300://Error
		iStateModbus_CP := iStateModbusError;
		timDelay.IN := FALSE;
		fbMBRead_FC3.bExecute := FALSE;
		fbMBWrite_FC16.bExecute := FALSE;
		bMBTCPError := TRUE; 		
		//Restart from new with the Read out part after an Error
		iStateModbusRead := 1;	
		iStateModbusError := 0;
		iStateModbusWrite := 0;
						
END_CASE

(*------------------------------------------------------------------------------------------Modbus TCP Functions---------------------------------------------------------------------------------------------*)

fbMBRead_FC3(	sIPAddr:= sIPAdress, 
				nTCPPort:= 502,
				cbLength:= SIZEOF(arrBuffer_FC3), 
				pDestAddr:= ADR(arrBuffer_FC3), 
				tTimeout:= T#5S );

FPError_FC_3(CLK:= fbMBRead_FC3.bError, Q=> );		

fbMBWrite_FC16(	sIPAddr:= sIPAdress, 
				nTCPPort:= 502, 
				cbLength:= SIZEOF(arrBuffer_FC16), 
				pSrcAddr:= ADR(arrBuffer_FC16), 
				tTimeout:= T#5S);	

FPError_FC_16(CLK:= fbMBWrite_FC16.bError, Q=> );

(*-----------------------------------------------------------Handle data to Global structure for electric charging stations-----------------------------------------------------------------*)

//Delte al old Data on GVL after a online change or change on the variable diNrOfEMS_IDOD
IF diNrOfEMS_IN <> diNrOfEMS_IN_CP AND iStateGVLData = 0 THEN iStateGVLData := 10; END_IF 

CASE iStateGVLData OF
	
	0://Init Step
		byWaitInStep := 0;
		diCounterForGVL := 1;
	
	1://Wait for 4 Steps before clean al Data on GVL
		byWaitInStep := byWaitInStep + 1;
		IF byWaitInStep >= 4 AND fbNumberDevice.bNumberIsCalculatet THEN iStateGVLData := 2; END_IF
		//To much Devices, back to the Init step
		IF byWaitInStep >= 4 AND NOT fbNumberDevice.bNumberIsCalculatet THEN iStateGVLData := 0; END_IF	
			
	2://Clear all Data in GVL
		FOR diLPForGVL := 1 TO Constants_Energy.diMaxNumberOfEMS BY 1 DO 
			Lynus_Standards.GVL_Energy.stDataElectricChargingStations[diLPForGVL,diCounterForGVL].bEnabled := FALSE;
			Lynus_Standards.GVL_Energy.stDataElectricChargingStations[diLPForGVL,diCounterForGVL].bIsControllable := FALSE;
			Lynus_Standards.GVL_Energy.stDataElectricChargingStations[diLPForGVL,diCounterForGVL].byErrorWarning := 0;
			Lynus_Standards.GVL_Energy.stDataElectricChargingStations[diLPForGVL,diCounterForGVL].byPriority := 0;
			Lynus_Standards.GVL_Energy.stDataElectricChargingStations[diLPForGVL,diCounterForGVL].lrPower := 0;
			Lynus_Standards.GVL_Energy.stDataElectricChargingStations[diLPForGVL,diCounterForGVL].lrPowerConsumption := 0;
			Lynus_Standards.GVL_Energy.stDataElectricChargingStations[diLPForGVL,diCounterForGVL].lrPowerProduction := 0;
			Lynus_Standards.GVL_Energy.stDataElectricChargingStations[diLPForGVL,diCounterForGVL].rMaxPower := 0;
			Lynus_Standards.GVL_Energy.stDataElectricChargingStations[diLPForGVL,diCounterForGVL].byElectricFuseLine := 0;
			//Set also the target value from ems back here to 0 and not in EMS function because EMS is in Standy when we have a online change (Problem when we delete a ems function and make a online change)
			Lynus_Standards.GVL_Energy.stDataElectricChargingStations[diLPForGVL,diCounterForGVL].rTargetPowerEMS := 0;	
		END_FOR
		
		//Counter for ECS
		diCounterForGVL := diCounterForGVL + 1;
		diCounterForGVL := LIMIT(0,diCounterForGVL,Constants_Energy.diMaxNumberOfElectricChargingStations);
		//Back to the init step
		IF diCounterForGVL >= Constants_Energy.diMaxNumberOfElectricChargingStations THEN iStateGVLData := 0; END_IF

	10://Clear old Data on GVL 		
		Lynus_Standards.GVL_Energy.stDataElectricChargingStations[diNrOfEMS_IN_CP,diNrOfECS_OUT].bEnabled := FALSE;
		Lynus_Standards.GVL_Energy.stDataElectricChargingStations[diNrOfEMS_IN_CP,diNrOfECS_OUT].bIsControllable := FALSE;
		Lynus_Standards.GVL_Energy.stDataElectricChargingStations[diNrOfEMS_IN_CP,diNrOfECS_OUT].byErrorWarning := 0;
		Lynus_Standards.GVL_Energy.stDataElectricChargingStations[diNrOfEMS_IN_CP,diNrOfECS_OUT].byPriority := 0;
		Lynus_Standards.GVL_Energy.stDataElectricChargingStations[diNrOfEMS_IN_CP,diNrOfECS_OUT].lrPower := 0;
		Lynus_Standards.GVL_Energy.stDataElectricChargingStations[diNrOfEMS_IN_CP,diNrOfECS_OUT].lrPowerConsumption := 0;
		Lynus_Standards.GVL_Energy.stDataElectricChargingStations[diNrOfEMS_IN_CP,diNrOfECS_OUT].lrPowerProduction := 0;
		Lynus_Standards.GVL_Energy.stDataElectricChargingStations[diNrOfEMS_IN_CP,diNrOfECS_OUT].rMaxPower := 0;
		Lynus_Standards.GVL_Energy.stDataElectricChargingStations[diNrOfEMS_IN_CP,diNrOfECS_OUT].byElectricFuseLine := 0;
									
		diNrOfEMS_IN_CP := diNrOfEMS_IN;
		//Back to the init step
		iStateGVLData := 0;

END_CASE 	 

IF diNrOfECS_OUT > 0 AND fbNumberDevice.bNumberIsCalculatet AND diNrOfEMS_IN > 0 THEN
	Lynus_Standards.GVL_Energy.stDataElectricChargingStations[diNrOfEMS_IN,diNrOfECS_OUT].bEnabled := fbCS.stDataECSOut.bEnabled;
	Lynus_Standards.GVL_Energy.stDataElectricChargingStations[diNrOfEMS_IN,diNrOfECS_OUT].bIsControllable := TRUE;
	Lynus_Standards.GVL_Energy.stDataElectricChargingStations[diNrOfEMS_IN,diNrOfECS_OUT].byErrorWarning := fbCS.stDataECSOut.byErrorWarning;
	Lynus_Standards.GVL_Energy.stDataElectricChargingStations[diNrOfEMS_IN,diNrOfECS_OUT].byPriority := fbCS.stDataECSOut.byPriority;
	Lynus_Standards.GVL_Energy.stDataElectricChargingStations[diNrOfEMS_IN,diNrOfECS_OUT].lrPower := fbCS.stDataECSOut.lrTotalPower;
	Lynus_Standards.GVL_Energy.stDataElectricChargingStations[diNrOfEMS_IN,diNrOfECS_OUT].lrPowerConsumption := fbCS.stDataECSOut.lrTotalPowerConsumption;
	Lynus_Standards.GVL_Energy.stDataElectricChargingStations[diNrOfEMS_IN,diNrOfECS_OUT].lrPowerProduction := fbCS.stDataECSOut.lrTotalPowerProduction;
	Lynus_Standards.GVL_Energy.stDataElectricChargingStations[diNrOfEMS_IN,diNrOfECS_OUT].rMaxPower := fbCS.stDataECSOut.rMaxPower;	
	Lynus_Standards.GVL_Energy.stDataElectricChargingStations[diNrOfEMS_IN,diNrOfECS_OUT].byElectricFuseLine := byElectricFuseLine;
END_IF 

(*----------------------------------------------------------Save persistent data----------------------------------------------------------------*)

arrPD[1](lrValue:= BOOL_TO_LREAL(bEnable), bEventBasedActive=> );
arrPD[2](lrValue:= BOOL_TO_LREAL(bPowerDataInvers), bEventBasedActive=> );
arrPD[3](lrValue:= DINT_TO_LREAL(diNrOfEMS_IN), bEventBasedActive=> );
arrPD[4](lrValue:= DINT_TO_LREAL(diNrOfEM_IN_CS), bEventBasedActive=> );
arrPD[5](lrValue:= BOOL_TO_LREAL(stSetupECS.bManualyOn), bEventBasedActive=> );
arrPD[6](lrValue:= BOOL_TO_LREAL(stSetupECS.bOnEmergPowerOff), bEventBasedActive=> );
arrPD[7](lrValue:= BYTE_TO_LREAL(stSetupECS.byCSMinPower), bEventBasedActive=> );
arrPD[8](lrValue:= BYTE_TO_LREAL(stSetupECS.byDisableSOC), bEventBasedActive=> );
arrPD[9](lrValue:= BYTE_TO_LREAL(stSetupECS.byEnableSOC), bEventBasedActive=> );
arrPD[10](lrValue:= BYTE_TO_LREAL(stSetupECS.byManualyTargetPower), bEventBasedActive=> );
arrPD[11](lrValue:= BYTE_TO_LREAL(stSetupECS.byPriority), bEventBasedActive=> );
arrPD[12](lrValue:= REAL_TO_LREAL(stSetupECS.rMaxPower), bEventBasedActive=> );
arrPD[13](lrValue:= DINT_TO_LREAL(diNrOfEMS_IN_CP), bEventBasedActive=> );
arrPD[14](lrValue:= BYTE_TO_LREAL(byElectricFuseLine), bEventBasedActive=> );
fbPDString(sText:= sIPAdress, bEventBasedActive=> );

END_FUNCTION_BLOCK

// ---- FBs/Siemens/FB_PAC2200.TcPOU
FUNCTION_BLOCK FB_PAC2200
VAR_INPUT PERSISTENT
	m_Enable					: BOOL;						//Enable the Fuctionblock and his logic
	str_IPAdress				: STRING(15);				//IP Adress of the meter
END_VAR
VAR_OUTPUT
	real_RealPower_kW				: REAL;					// Real power in W
	real_RealPowerL1_kW				: REAL;					// Real power in W
	real_RealPowerL2_kW				: REAL;					// Real power in W
	real_RealPowerL3_kW				: REAL;					// Real power in W
	real_ReactivePower_kVAr			: REAL;					// Reactive power in VAr
	real_ApparentPower_kVA			: REAL;					// Apparent power in VA
	real_Frequency_Hz				: REAL;					// Frequency in Hz
	real_VoltageL1N_V				: REAL;					//  Voltage L1-N in V 
	real_VoltageL2N_V				: REAL;					//  Voltage L2-N in V 
	real_VoltageL3N_V				: REAL;					//  Voltage L3-N in V 
	real_VoltageL1L2_V				: REAL;					//  Voltage L1-L2 in V 
	real_VoltageL2L3_V				: REAL;					//  Voltage L2-L3 in V 
	real_VoltageL3L1_V				: REAL;					//  Voltage L3-L1 in V 
	real_CurrentL1_A				: REAL;					//  Current L1 in A
	real_CurrentL2_A				: REAL;					//  Current L2 in A
	real_CurrentL3_A				: REAL;					//  Current L3 in A
	real_EnergyTotal_Import_T1_kWh	: REAL;					// Energy total in Wh
	real_EnergyTotal_Import_T2_kWh	: REAL;					// Energy total in Wh
	real_EnergyTotal_Export_T1_kWh	: REAL;					// Energy total in Wh
	real_EnergyTotal_Export_T2_kWh	: REAL;					// Energy total in Wh
	
	m_PollSuccessful				: BOOL;					// Poll succesfull		
	udint_Error_ID					: UDINT;				// ERR ID FB_MBReadRegs
END_VAR
VAR
//	{attribute 'hide'}
	w_Adress					: WORD;						//modbus adress
//	{attribute 'hide'}
	usint_Quantity				: USINT;					//Number of Words to get polled, max 100
//	{attribute 'hide'}
	fb_Convert_Data				: FB_Convert_Dword_Real;
//	{attribute 'hide'}
	e_ByteOrderConvert	: eByteOrder;						//Byte Format
//	{attribute 'hide'}
	timer_Delay					: TON;						//Timer for Delay between Requests
//	{attribute 'hide'}
	timer_DelayStart			: TON;						//Timer to start the state machine with Delay after enabling or after the system ist restartet
//	{attribute 'hide'}
	timer_TimeOut				: TON;						//Timer for Timeout MB Read
//	{attribute 'hide'}
	iStateModbusRead			: INT;						//State machine for read out Data over Modbus RTU
//	{attribute 'hide'}
	fbMBRead_FC3				: FB_MBReadRegs  ;		//Modbus Read Function (FC3)
//	{attribute 'hide'}
	ftrig_PEnable				: f_trig;					//Internal positive Edge
//	{attribute 'hide'}
	iStateModbusError			: INT;						//State machine for error out Data over Modbus TCP/IP	
//	{attribute 'hide'}
	FPError_FC_3				: R_TRIG;					//Internal positive Edge
//	{attribute 'hide'}
	arrBuffer_FC3				: ARRAY[0..100] OF WORD;		//Buffer with Data from FC3
//	{attribute 'hide'}
	arrBuffer_Received			: ARRAY[1..2,0..100] OF WORD;		//Total received Data
//	{attribute 'hide'}
	timer_Connection_ok			: TON;
//	{attribute 'hide'}
	int_Data_Received			: INT;
//	{attribute 'hide'}
	m_MBTCPError				: BOOL;
//	{attribute 'hide'}
	int_Data_Received_old		: INT;
//	{attribute 'hide'}
	timer_Connection_ok_TOF	: TOF;
//	{attribute 'hide'}
	m_Poll_ok: BOOL;
//	{attribute 'hide'}
	timer_Wait: Ton;
//	{attribute 'hide'}
	int_TimeoutError: INT;
//	{attribute 'hide'}
	int_FC4Error: INT;
//	{attribute 'hide'}
	i: INT;
//	{attribute 'hide'}
	x: INT;

END_VAR

// v0.1 by Stefan Lackner 20230714
// reads out Siemens PC2200 Multimeters


(*--------------------------------------------------------------------------------------------Limits-------------------------------------------------------------------------------------*)
w_Adress := LIMIT(0,w_Adress,65000);
usint_Quantity := LIMIT(1,usint_Quantity,100);
	
(*--------------------------------------------------------------------------------------------State Machine Read--------------------------------------------------------------------------------------*)

//Timer for Delay
timer_Delay(IN:= , PT:= T#50MS, Q=> , ET=> );

//Timeout Timer is dissabled when the Init Step is aktiv or the function is not enabled
IF iStateModbusRead = 0 OR NOT m_Enable THEN 
	timer_Timeout.IN := FALSE; 
END_IF
timer_Timeout(IN:= , PT:= T#1S, Q=> , ET=> );

//Enable with Delay that not all sockets have to be created at the same time
timer_DelayStart(IN:= m_Enable, PT:= T#1S, Q=> , ET=> );
ftrig_PEnable(CLK:= timer_DelayStart.Q, Q=> );

IF ftrig_PEnable.Q AND iStateModbusRead = 0 THEN 
	iStateModbusRead := 1; 
END_IF		
		
//Not Enabled
IF NOT m_Enable THEN 
	iStateModbusRead := 0; 
	iStateModbusError := 0; 
END_IF		
		
CASE iStateModbusRead OF

	0://Init Step 
		timer_Delay.IN := FALSE;
		fbMBRead_FC3.bExecute := FALSE;
		m_Poll_ok:=FALSE;
		int_Data_Received:=0;
		iStateModbusRead := iStateModbusRead+1;

	1: // clean the array  Poll 1
		FOR i:=0 TO 100 BY 1 DO
			arrBuffer_FC3[i] := 0;
		END_FOR
		w_Adress := 1;
		usint_Quantity := 100; 
		iStateModbusRead := iStateModbusRead+1;
		
	2://read the required registers
		//Start Read Poll 1
		fbMBRead_FC3.nQuantity := usint_Quantity;
		fbMBRead_FC3.nMBAddr := w_Adress;
		fbMBRead_FC3.bExecute := TRUE;
		fbMBRead_FC3.nUnitID := 1;
		timer_Timeout.IN := TRUE;
		IF fbMBRead_FC3.bBusy THEN 
			timer_Delay.IN := TRUE; 
		END_IF
		
		//Wait for Delay, copy Data and then next step
		IF NOT fbMBRead_FC3.bBusy AND NOT fbMBRead_FC3.bError AND timer_Delay.Q THEN
			m_Poll_ok:=TRUE;
			int_Data_Received:=int_Data_Received+1;
			m_MBTCPError := FALSE; 
			
			FOR i:=0 TO 100 BY 1 DO
				arrBuffer_Received[1,i] := arrBuffer_FC3[i];
			END_FOR
			
			//Go to Next Step
			timer_Timeout.IN := FALSE;
			fbMBRead_FC3.bExecute := FALSE;
			timer_Delay.IN := FALSE;		
			iStateModbusRead := iStateModbusRead+1;
		END_IF	

		//Error or Timeout
		IF FPError_FC_3.Q THEN 
			iStateModbusError := 300;
			int_FC4Error := int_FC4Error+1;
		ELSIF timer_Timeout.Q THEN  
			timer_Timeout.IN := FALSE; 	
			iStateModbusError := 300;
			int_TimeoutError := int_TimeoutError+1;
		END_IF
	
	3://Wait and go to next step
		timer_Wait.IN := TRUE;
		
		IF timer_Wait.Q = TRUE THEN
			iStateModbusRead := iStateModbusRead+1;
			timer_Wait.IN :=FALSE;
		END_IF

	4: // clean the array  Poll 2
		FOR i:=0 TO 100 BY 1 DO
			arrBuffer_FC3[i] := 0;
		END_FOR
		w_Adress := 2801;;
		usint_Quantity := 10; 
		iStateModbusRead := iStateModbusRead+1;
		
	5://read the required registers
		//Start Read Poll 2
		fbMBRead_FC3.nQuantity := usint_Quantity;
		fbMBRead_FC3.nMBAddr := w_Adress;
		fbMBRead_FC3.bExecute := TRUE;
		fbMBRead_FC3.nUnitID := 1;
		timer_Timeout.IN := TRUE;
		IF fbMBRead_FC3.bBusy THEN 
			timer_Delay.IN := TRUE; 
		END_IF
		
		//Wait for Delay, copy Data and then next step
		IF NOT fbMBRead_FC3.bBusy AND NOT fbMBRead_FC3.bError AND timer_Delay.Q THEN
			m_Poll_ok:=TRUE;
			int_Data_Received:=int_Data_Received+1;
			m_MBTCPError := FALSE; 
			
			FOR i:=0 TO 9 BY 1 DO
				arrBuffer_Received[2,i] := arrBuffer_FC3[i];
			END_FOR
			
			//Go to Next Step
			timer_Timeout.IN := FALSE;
			fbMBRead_FC3.bExecute := FALSE;
			timer_Delay.IN := FALSE;		
			iStateModbusRead := iStateModbusRead+1;
		END_IF	

		//Error or Timeout
		IF FPError_FC_3.Q THEN 
			iStateModbusError := 300;
			int_FC4Error := int_FC4Error+1;
		ELSIF timer_Timeout.Q THEN  
			timer_Timeout.IN := FALSE; 	
			iStateModbusError := 300;
			int_TimeoutError := int_TimeoutError+1;
		END_IF
	
	6://Wait and go to next step
		timer_Wait.IN := TRUE;
		
		IF timer_Wait.Q = TRUE THEN
			iStateModbusRead := 30;
			timer_Wait.IN :=FALSE;
		END_IF
		

	
	30: // convert data
		e_ByteOrderConvert := 0;
		x:=0;
		fb_Convert_Data(	word_In_1:= arrBuffer_Received[1,x], 
							word_In_2:= arrBuffer_Received[1,x+1], 
							e_ByteOrderIn:= e_ByteOrderConvert, 
							real_Output=> real_VoltageL1N_V);
		x:=x+2;
		fb_Convert_Data(	word_In_1:= arrBuffer_Received[1,x], 
							word_In_2:= arrBuffer_Received[1,x+1], 
							e_ByteOrderIn:= e_ByteOrderConvert, 
							real_Output=> real_VoltageL2N_V);
		x:=x+2;
		fb_Convert_Data(	word_In_1:= arrBuffer_Received[1,x], 
							word_In_2:= arrBuffer_Received[1,x+1], 
							e_ByteOrderIn:= e_ByteOrderConvert, 
							real_Output=> real_VoltageL3N_V);		
		x:=x+2;
		fb_Convert_Data(	word_In_1:= arrBuffer_Received[1,x], 
							word_In_2:= arrBuffer_Received[1,x+1], 
							e_ByteOrderIn:= e_ByteOrderConvert, 
							real_Output=> real_VoltageL1L2_V);
		x:=x+2;
		fb_Convert_Data(	word_In_1:= arrBuffer_Received[1,x], 
							word_In_2:= arrBuffer_Received[1,x+1], 
							e_ByteOrderIn:= e_ByteOrderConvert, 
							real_Output=> real_VoltageL2L3_V);
		x:=x+2;
		fb_Convert_Data(	word_In_1:= arrBuffer_Received[1,x], 
							word_In_2:= arrBuffer_Received[1,x+1], 
							e_ByteOrderIn:= e_ByteOrderConvert, 
							real_Output=> real_VoltageL3L1_V);
		x:=x+2;
		fb_Convert_Data(	word_In_1:= arrBuffer_Received[1,x], 
							word_In_2:= arrBuffer_Received[1,x+1], 
							e_ByteOrderIn:= e_ByteOrderConvert, 
							real_Output=> real_CurrentL1_A);
		x:=x+2;
		fb_Convert_Data(	word_In_1:= arrBuffer_Received[1,x], 
							word_In_2:= arrBuffer_Received[1,x+1], 
							e_ByteOrderIn:= e_ByteOrderConvert, 
							real_Output=> real_CurrentL2_A);
		x:=x+2;
		fb_Convert_Data(	word_In_1:= arrBuffer_Received[1,x], 
							word_In_2:= arrBuffer_Received[1,x+1], 
							e_ByteOrderIn:= e_ByteOrderConvert, 
							real_Output=> real_CurrentL3_A);		
		x:=24;
		fb_Convert_Data(	word_In_1:= arrBuffer_Received[1,x], 
							word_In_2:= arrBuffer_Received[1,x+1], 
							e_ByteOrderIn:= e_ByteOrderConvert, 
							real_Output=> real_RealPowerL1_kW);
							real_RealPowerL1_kW := real_RealPowerL1_kW/1000;
		x:=x+2;		
		fb_Convert_Data(	word_In_1:= arrBuffer_Received[1,x], 
							word_In_2:= arrBuffer_Received[1,x+1], 
							e_ByteOrderIn:= e_ByteOrderConvert, 
							real_Output=> real_RealPowerL2_kW);		
							real_RealPowerL2_kW := real_RealPowerL2_kW/1000;
		x:=x+2;		
		fb_Convert_Data(	word_In_1:= arrBuffer_Received[1,x], 
							word_In_2:= arrBuffer_Received[1,x+1], 
							e_ByteOrderIn:= e_ByteOrderConvert, 
							real_Output=> real_RealPowerL3_kW);
							real_RealPowerL3_kW := real_RealPowerL3_kW/1000;								
		x:=54;		
		fb_Convert_Data(	word_In_1:= arrBuffer_Received[1,x], 
							word_In_2:= arrBuffer_Received[1,x+1], 
							e_ByteOrderIn:= e_ByteOrderConvert, 
							real_Output=> real_Frequency_Hz);									
		x:=62;		
		fb_Convert_Data(	word_In_1:= arrBuffer_Received[1,x], 
							word_In_2:= arrBuffer_Received[1,x+1], 
							e_ByteOrderIn:= e_ByteOrderConvert, 
							real_Output=> real_ApparentPower_kVA);
							real_ApparentPower_kVA := real_ApparentPower_kVA/1000;									
		x:=x+2;	
		fb_Convert_Data(	word_In_1:= arrBuffer_Received[1,x], 
							word_In_2:= arrBuffer_Received[1,x+1], 
							e_ByteOrderIn:= e_ByteOrderConvert, 
							real_Output=> real_RealPower_kW);	
							real_RealPower_kW := real_RealPower_kW/1000;
		x:=x+2;	
		fb_Convert_Data(	word_In_1:= arrBuffer_Received[1,x], 
							word_In_2:= arrBuffer_Received[1,x+1], 
							e_ByteOrderIn:= e_ByteOrderConvert, 
							real_Output=> real_ReactivePower_kVAr);	
							real_ReactivePower_kVAr := real_ReactivePower_kVAr/1000;
		//2nd Poll
		x:=0;	
		fb_Convert_Data(	word_In_1:= arrBuffer_Received[2,x], 
							word_In_2:= arrBuffer_Received[2,x+1], 
							e_ByteOrderIn:= e_ByteOrderConvert, 
							real_Output=> real_EnergyTotal_Import_T1_kWh);		
							real_EnergyTotal_Import_T1_kWh := real_EnergyTotal_Import_T1_kWh/1000;
		x:=x+2;	
		fb_Convert_Data(	word_In_1:= arrBuffer_Received[2,x], 
							word_In_2:= arrBuffer_Received[2,x+1], 
							e_ByteOrderIn:= e_ByteOrderConvert, 
							real_Output=> real_EnergyTotal_Import_T2_kWh);		
							real_EnergyTotal_Import_T2_kWh := real_EnergyTotal_Import_T2_kWh/1000;
		x:=x+2;	
		fb_Convert_Data(	word_In_1:= arrBuffer_Received[2,x], 
							word_In_2:= arrBuffer_Received[2,x+1], 
							e_ByteOrderIn:= e_ByteOrderConvert, 
							real_Output=> real_EnergyTotal_Export_T1_kWh);	
							real_EnergyTotal_Export_T1_kWh := real_EnergyTotal_Export_T1_kWh/1000;	
		x:=x+2;	
		fb_Convert_Data(	word_In_1:= arrBuffer_Received[2,x], 
							word_In_2:= arrBuffer_Received[2,x+1], 
							e_ByteOrderIn:= e_ByteOrderConvert, 
							real_Output=> real_EnergyTotal_Export_T2_kWh);		
							real_EnergyTotal_Export_T2_kWh := real_EnergyTotal_Export_T2_kWh/1000;							

		
		// go to next state
		iStateModbusRead := iStateModbusRead+1;		
		
	31://Wait and go to start
		timer_Wait.IN := TRUE;
		
		IF timer_Wait.Q = TRUE THEN
			iStateModbusRead := 1;
			timer_Wait.IN :=FALSE;
		END_IF	

END_CASE

(* wait timer*)

timer_Wait(PT:=T#1S);


(*------------------------------------------------------------------Error and Warning----------------------------------------------------------------------------*)	
 
timer_Connection_ok			(In:=int_Data_Received<>int_Data_Received_old,PT:=T#10S);
timer_Connection_ok_TOF		(In:=NOT(int_Data_Received<>int_Data_Received_old) AND int_Data_Received>3 ,PT:=T#20S);
int_Data_Received_old:=int_Data_Received;
m_PollSuccessful:=NOT timer_Connection_ok.Q AND timer_Connection_ok_TOF.Q ;

(*------------------------------------------------------------------------------------------Modbus TCP Functions---------------------------------------------------------------------------------------------*)

fbMBRead_FC3(	sIPAddr:= str_IPAdress, 
				nTCPPort:= 502,
				cbLength:= SIZEOF(arrBuffer_FC3), 
				pDestAddr:= ADR(arrBuffer_FC3), 
				tTimeout:= T#10S,
				nErrId => udint_Error_ID);

FPError_FC_3(CLK:= fbMBRead_FC3.bError, Q=> );		

(*------------------------------------------------------------------------------------------State Machine Error---------------------------------------------------------------------------------------------*)	

CASE iStateModbusError OF
	
	300://Error
		timer_Wait.IN :=TRUE;
		timer_Delay.IN := FALSE;
		fbMBRead_FC3.bExecute := FALSE;
		m_MBTCPError := TRUE; 		
		m_Poll_ok:=FALSE;
		int_Data_Received:=0;
		
				//Restart from new with the Read out part after an Error
		IF timer_Wait.Q = TRUE THEN
			iStateModbusRead := 0;	
			iStateModbusError := 0;
			timer_Wait.IN :=FALSE;
			timer_Timeout.IN := FALSE;
		END_IF		
							
END_CASE

END_FUNCTION_BLOCK

// ---- FBs/SolarEdge/FB_SunSpec_PV_Inverter.TcPOU
// {attribute 'hide_all_locals'}
FUNCTION_BLOCK FB_SunSpec_PV_Inverter
VAR_INPUT PERSISTENT
	bEnable						: BOOL;												//True = Function is enabled, FALSE = Function is dissabled, no new Data
	sIPAdress					: STRING(15);										//IP Adress from the Inverter
	byUnitID_Inverter			: BYTE;												//Unit ID from the Inverter (1 to 247)
END_VAR
VAR_OUTPUT
	stDataSunSpec				: ST_SunSpec_PV_OutData;							//Output structure with Data from SunSpec
	stDataEMPower_PV			: ST_ElectricMeter_Output_Power;					//Output structure with Data from Electric Meter PV (Power Data)
	stDataEMCounter_PV			: ST_ElectricMeter_Output_Counter;					//Output structure with Data from Electric Meter PV (Counter Data)
	diNrOfEM_OUT_PV				: DINT;												//Active Number from the Electric Meter for using on other functions
END_VAR
VAR
	fbElMeter					: FB_ElectricMeter;									//Electric Meter Function 
	fbNumberDevice				: FB_NumberOfDevice;								//Function block to calcualte the number of the Device
	fbConvertEnergyRegister		: FB_CV_WORD_TO_DWORD;								//Convert function
	fbMBRead_FC3				: FB_MBReadRegs;									//Modbus Read Function (FC3)
	timDelay					: TON;												//Timer for Delay between Requests
	timTimeout					: TON;												//Timer for Timeout
	timDissableFunctions		: TON;												//Timer to dissable the Function after Lynus_Standards.Constants_General.tTimeDissableLynusFunctions Days without connection to the Lynus Cloud
	timResetConnectionOnGVL		: TON;												//Timer to try reset the connection Flag on the GVL. (When somebody delete the Connection Function and make only a onlinechange)
	FPEnable					: R_TRIG;											//Internal positive Edge
	FPError_FC_3				: R_TRIG;											//Internal positive Edge
	PD_String					: FB_PersistentData_String;							//Function to save persistent data 
	stFloat						: ST_UN_FLOAT_CONVERT_DWORD_REAL;					//Convert the Float Raw Value
	arrBuffer_FC3				: ARRAY[1..125] OF WORD;							//Buffer with Data from FC3
	arrPD						: ARRAY[1..2] OF FB_PersistentData_Number;			//Function to save persistent data 
	byWaitInStep				: BYTE;												//Wait in Step before start to clean data on PLC
	iStateGVLData				: INT;												//State machine to handle the data on the GVL
	iStateModbus				: INT;												//State variable for Statemachine
	iStateModbus_CP				: INT;												//Compare State variable
	diCounterForGVL				: DINT;												//Counter to clean old data on GVL
	lrCheckValue				: LREAL;											//Internal Value to check the value before convert
	lrTemp: LREAL;
	FB_word_to_dword: FB_CV_WORD_TO_DWORD;
	x: eByteOrder;
END_VAR

//Creator : Stefan Lackner
//Company : EfficientIO
//Date : 27.09.2022
//Version : 0.0.0.1		--> not tested yet!

//With this function its possible to read out values from the SunSpec from the manufacturer SolarEdge
//This Function read out the Values from 1 SunSpec inverter
//The protocol to the Inverter is Modbus TCP
//Attention. To access the registers, an offset of 1 must always be subtracted. Register 40001 would then be on register 40000.
//The document "sunspec-implementation-technical-note.pdf" version 2.4 got used for the Modbus adress List

//NOTE for diNr.....Designation => 
//_IN = Here Data come in from other Functions or go out to other functions about the GVL
//_OUT = Here Data go out to other functions about the GVL

(*------------------------------------------------------------------------------------------General Input Part---------------------------------------------------------------------------------------------*)

//Check limitation
byUnitID_Inverter := LIMIT(1,byUnitID_Inverter,247);

(*-------------------------------------------------------------Calcualte the number of EM System---------------------------------------------------------------*)

fbNumberDevice(
	diActualNumberOfDevices:= Lynus_Standards.GVL_Energy.stNumberOfDevices.diNumberOfElectricMeters, 
	diMaxNumberOfDevices:= Constants_Energy.diMaxNumberOfElectricMeters, 
	udiCounterOnlineChange:= TwinCAT_SystemInfoVarList._AppInfo.OnlineChangeCnt, 
	bNumberIsCalculatet=> , 
	bFPNumberIsCalculatet=> , 
	bOnlineChange=> , 
	diNumberForThisDevice=> diNrOfEM_OUT_PV, 
	diNumberOfTotalDevices=> );

//Write new Numer on GVL
IF fbNumberDevice.bFPNumberIsCalculatet THEN
	Lynus_Standards.GVL_Energy.stNumberOfDevices.diNumberOfElectricMeters := fbNumberDevice.diNumberOfTotalDevices;	
END_IF 

//Delete old Number on GVL
IF fbNumberDevice.bOnlineChange THEN 
	Lynus_Standards.GVL_Energy.stNumberOfDevices.diNumberOfElectricMeters := diNrOfEM_OUT_PV;	
		iStateGVLData := 1; 
END_IF

(*-------------------------------------------------------------Service from Backend is ready and check the connection to backend for dissabel/enable Function---------------------------------------------------------------*)

//Try to reset the variable for connection on the GVL. When all is normal then the EfficientIO Mqtt connection function set this variable to true in the next cycle
//When we have no connection to the backend then after Lynus_Standards.Constants_General.tTimeDissableLynusFunctions days the Function is dissabled with all of his functionalities
timResetConnectionOnGVL(IN:= NOT timResetConnectionOnGVL.Q, PT:= T#1H, Q=> , ET=> );
IF timResetConnectionOnGVL.Q THEN 
	Lynus_Standards.GVL_Communicator.bStateConnectionToEnableFunctions := FALSE; 
END_IF
IF NOT Lynus_Standards.GVL_Communicator.bStateConnectionToEnableFunctions THEN 
	timDissableFunctions.IN := TRUE; 
ELSE 
	timDissableFunctions.IN := FALSE; 
END_IF  
timDissableFunctions(IN:= , PT:= Lynus_Standards.Constants_General.tTimeDissableLynusFunctions, Q=> , ET=> );
	
(*------------------------------------------------------------------------------------------State Machine---------------------------------------------------------------------------------------------*)
	
//Enable
FPEnable(CLK:= bEnable, Q=> );
IF FPEnable.Q AND iStateModbus = 0 THEN 
	iStateModbus := 1; 
END_IF
IF NOT bEnable OR timDissableFunctions.Q THEN 
	iStateModbus := 0; 
END_IF

//Timer for delay
timDelay(IN:= , PT:= T#100MS, Q=> , ET=> );	

//Timer for Timeout in Statemachine
IF iStateModbus = iStateModbus_CP THEN 
	timTimeout.IN := TRUE; 
ELSE 
	timTimeout.IN := FALSE; 
END_IF
IF iStateModbus = 0 THEN 
	timTimeout.IN := FALSE; 
END_IF
timTimeout(IN:= , PT:= T#20S, Q=> , ET=> );	

//Statemachine
CASE iStateModbus OF
	
	0://Init Step
		iStateModbus_CP := iStateModbus;
		timDelay.IN := FALSE;
		
		stDataSunSpec.bFunctionIsActive := FALSE;
		stDataSunSpec.eOperatingStateInverter := E_SunSpec_PV_OperatingState.eNoDataReceived;
		fbMBRead_FC3.bExecute := FALSE;
		lrCheckValue := 0;
									
	1://Read out first Registers from 40001 to 40109
		stDataSunSpec.bFunctionIsActive := TRUE;
		iStateModbus_CP := iStateModbus;
		
		fbMBRead_FC3.nQuantity := 108;
		fbMBRead_FC3.nMBAddr := 40000;  
		fbMBRead_FC3.bExecute := TRUE;
		fbMBRead_FC3.nUnitID := byUnitID_Inverter;
			
		IF fbMBRead_FC3.bBusy THEN 
			timDelay.IN := TRUE; 
		END_IF
		
		//Wait for Delay, copy Data and then next step
		IF NOT fbMBRead_FC3.bBusy AND NOT fbMBRead_FC3.bError AND timDelay.Q AND fbMBRead_FC3.nErrId=0 AND fbMBRead_FC3.cbRead<>0 THEN
			//Copy Data Current L1
			lrCheckValue := (UINT_TO_LREAL(WORD_TO_UINT(arrBuffer_FC3[73]))*EXPT(10,(WORD_TO_INT(arrBuffer_FC3[76]))));
					//fbConvertEnergyRegister(wInputValue_1:= arrBuffer_FC3[3], wInputValue_2:= arrBuffer_FC3[4], eByteOrderForConvert:= eByteOrder.eBigEndian, dwOutputValue=> );
					//stFloat.dwRawValue := fbConvertEnergyRegister.dwOutputValue;
					//lrCheckValue := stFloat.rValueFloat;	
			IF lrCheckValue >= - 3.402823E+38 AND lrCheckValue <= 3.402823E+38 THEN 
				fbElMeter.lrCurrentL1 := lrCheckValue;
			ELSE
				iStateModbus := 300;
				stDataSunSpec.eErrorState := E_SunSpec_PV_Error.eSunSpecTooBigValueReceived;		
			END_IF
			//Copy Data Current L2
			lrCheckValue := (UINT_TO_LREAL(WORD_TO_UINT(arrBuffer_FC3[74]))*EXPT(10,(WORD_TO_INT(arrBuffer_FC3[76]))));
			IF lrCheckValue >= - 3.402823E+38 AND lrCheckValue <= 3.402823E+38 THEN 
				fbElMeter.lrCurrentL2 := lrCheckValue;
			ELSE
				iStateModbus := 300;
				stDataSunSpec.eErrorState := E_SunSpec_PV_Error.eSunSpecTooBigValueReceived;		
			END_IF
			//Copy Data Current L3
			lrCheckValue := (UINT_TO_LREAL(WORD_TO_UINT(arrBuffer_FC3[75]))*EXPT(10,(WORD_TO_INT(arrBuffer_FC3[76]))));
			IF lrCheckValue >= - 3.402823E+38 AND lrCheckValue <= 3.402823E+38 THEN 
				fbElMeter.lrCurrentL3 := lrCheckValue;
			ELSE
				iStateModbus := 300;
				stDataSunSpec.eErrorState := E_SunSpec_PV_Error.eSunSpecTooBigValueReceived;		
			END_IF
			//Copy Data Voltage L1-L2
			lrCheckValue := (UINT_TO_LREAL(WORD_TO_UINT(arrBuffer_FC3[77]))*EXPT(10,(WORD_TO_INT(arrBuffer_FC3[83]))));
			IF lrCheckValue >= - 3.402823E+38 AND lrCheckValue <= 3.402823E+38 THEN 
				fbElMeter.lrVoltageL1L2 := lrCheckValue;
			ELSE
				iStateModbus := 300;
				stDataSunSpec.eErrorState := E_SunSpec_PV_Error.eSunSpecTooBigValueReceived;		
			END_IF
			//Copy Data Voltage L2-L3
			lrCheckValue := (UINT_TO_LREAL(WORD_TO_UINT(arrBuffer_FC3[78]))*EXPT(10,(WORD_TO_INT(arrBuffer_FC3[83]))));
			IF lrCheckValue >= - 3.402823E+38 AND lrCheckValue <= 3.402823E+38 THEN 
				fbElMeter.lrVoltageL2L3 := lrCheckValue;
			ELSE
				iStateModbus := 300;
				stDataSunSpec.eErrorState := E_SunSpec_PV_Error.eSunSpecTooBigValueReceived;		
			END_IF
			//Copy Data Voltage L3-L1
			lrCheckValue := (UINT_TO_LREAL(WORD_TO_UINT(arrBuffer_FC3[79]))*EXPT(10,(WORD_TO_INT(arrBuffer_FC3[83]))));
			IF lrCheckValue >= - 3.402823E+38 AND lrCheckValue <= 3.402823E+38 THEN 
				fbElMeter.lrVoltageL3L1 := lrCheckValue;
			ELSE
				iStateModbus := 300;
				stDataSunSpec.eErrorState := E_SunSpec_PV_Error.eSunSpecTooBigValueReceived;		
			END_IF
			//Copy Data Voltage L1-N
			lrCheckValue := (UINT_TO_LREAL(WORD_TO_UINT(arrBuffer_FC3[80]))*EXPT(10,(WORD_TO_INT(arrBuffer_FC3[83]))));
			IF lrCheckValue >= - 3.402823E+38 AND lrCheckValue <= 3.402823E+38 THEN 
				fbElMeter.lrVoltageL1N := lrCheckValue;
			ELSE
				iStateModbus := 300;
				stDataSunSpec.eErrorState := E_SunSpec_PV_Error.eSunSpecTooBigValueReceived;		
			END_IF
			//Copy Data Voltage L2-N
			lrCheckValue := (UINT_TO_LREAL(WORD_TO_UINT(arrBuffer_FC3[81]))*EXPT(10,(WORD_TO_INT(arrBuffer_FC3[83]))));
			IF lrCheckValue >= - 3.402823E+38 AND lrCheckValue <= 3.402823E+38 THEN 
				fbElMeter.lrVoltageL2N := lrCheckValue;
			ELSE
				iStateModbus := 300;
				stDataSunSpec.eErrorState := E_SunSpec_PV_Error.eSunSpecTooBigValueReceived;		
			END_IF
			//Copy Data Voltage L3-N
			lrCheckValue := (UINT_TO_LREAL(WORD_TO_UINT(arrBuffer_FC3[82]))*EXPT(10,(WORD_TO_INT(arrBuffer_FC3[83]))));
			IF lrCheckValue >= - 3.402823E+38 AND lrCheckValue <= 3.402823E+38 THEN 
				fbElMeter.lrVoltageL3N := lrCheckValue;
			ELSE
				iStateModbus := 300;
				stDataSunSpec.eErrorState := E_SunSpec_PV_Error.eSunSpecTooBigValueReceived;		
			END_IF
			//Copy Data AC Power
			lrCheckValue := (UINT_TO_LREAL(WORD_TO_UINT(arrBuffer_FC3[84]))*EXPT(10,(WORD_TO_INT(arrBuffer_FC3[85]))));
			IF lrCheckValue >= - 3.402823E+38 AND lrCheckValue <= 3.402823E+38 THEN 
				fbElMeter.lrPowerTotal := lrCheckValue;
			ELSE
				iStateModbus := 300;
				stDataSunSpec.eErrorState := E_SunSpec_PV_Error.eSunSpecTooBigValueReceived;		
			END_IF
			//Copy Data Frequency
			lrCheckValue := (UINT_TO_LREAL(WORD_TO_UINT(arrBuffer_FC3[86]))*EXPT(10,(WORD_TO_INT(arrBuffer_FC3[87]))));
			IF lrCheckValue >= - 3.402823E+38 AND lrCheckValue <= 3.402823E+38 THEN 
				fbElMeter.lrFrequency := lrCheckValue;
			ELSE
				iStateModbus := 300;
				stDataSunSpec.eErrorState := E_SunSpec_PV_Error.eSunSpecTooBigValueReceived;		
			END_IF			
			//Copy Data Apparent Power
			lrCheckValue := (UINT_TO_LREAL(WORD_TO_UINT(arrBuffer_FC3[88]))*EXPT(10,(WORD_TO_INT(arrBuffer_FC3[89]))));
			IF lrCheckValue >= - 3.402823E+38 AND lrCheckValue <= 3.402823E+38 THEN 
				fbElMeter.lrApparentPowerTotal := lrCheckValue;
			ELSE
				iStateModbus := 300;
				stDataSunSpec.eErrorState := E_SunSpec_PV_Error.eSunSpecTooBigValueReceived;		
			END_IF			
			//Copy Data Reactive Power
			lrCheckValue := (UINT_TO_LREAL(WORD_TO_UINT(arrBuffer_FC3[90]))*EXPT(10,(WORD_TO_INT(arrBuffer_FC3[91]))));
			IF lrCheckValue >= - 3.402823E+38 AND lrCheckValue <= 3.402823E+38 THEN 
				fbElMeter.lrReactivePowerTotal := lrCheckValue;
			ELSE
				iStateModbus := 300;
				stDataSunSpec.eErrorState := E_SunSpec_PV_Error.eSunSpecTooBigValueReceived;		
			END_IF			
			//Copy Data AC production Energy
			FB_word_to_dword(	wInputValue_1 := arrBuffer_FC3[94],
								wInputValue_2 := arrBuffer_FC3[95],
								eByteOrderForConvert := x);
			lrCheckValue := DWORD_TO_LREAL(FB_word_to_dword.dwOutputValue)* EXPT(10,(WORD_TO_INT(arrBuffer_FC3[96])));
			IF lrCheckValue >= - 3.402823E+38 AND lrCheckValue <= 3.402823E+38 THEN 
				fbElMeter.lrCounterEnergyT1_Production := lrCheckValue / 1000;
			ELSE
				iStateModbus := 300;
				stDataSunSpec.eErrorState := E_SunSpec_PV_Error.eSunSpecTooBigValueReceived;		
			END_IF			
			//Operating State	
						(*I_STATUS_OFF			1 	Off
						I_STATUS_SLEEPING		2	Sleeping (auto-shutdown) – Night mode
						I_STATUS_STARTING		3	Grid Monitoring/wake-up
						I_STATUS_MPPT			4	Inverter is ON and producing power
						I_STATUS_THROTTLED		5	Production (curtailed)
						I_STATUS_SHUTTING_DOWN	6	Shutting down
						I_STATUS_FAULT			7	Fault
						I_STATUS_STANDBY		8	Maintenance/setup*)
	
			IF 			arrBuffer_FC3[108] = 1 THEN stDataSunSpec.eOperatingStateInverter := E_Symo_PV_OperatingState.eOff;
				ELSIF 	arrBuffer_FC3[108] = 2 THEN stDataSunSpec.eOperatingStateInverter := E_Symo_PV_OperatingState.eSleeping;
				ELSIF 	arrBuffer_FC3[108] = 3 THEN stDataSunSpec.eOperatingStateInverter := E_Symo_PV_OperatingState.eStartingUp;
				ELSIF 	arrBuffer_FC3[108] = 4 THEN stDataSunSpec.eOperatingStateInverter := E_Symo_PV_OperatingState.eTrackingPowerPoint;
				ELSIF 	arrBuffer_FC3[108] = 5 THEN stDataSunSpec.eOperatingStateInverter := E_Symo_PV_OperatingState.eForcedPowerReduction;
				ELSIF 	arrBuffer_FC3[108] = 6 THEN stDataSunSpec.eOperatingStateInverter := E_Symo_PV_OperatingState.eShuttingDown;
				ELSIF 	arrBuffer_FC3[108] = 7 THEN stDataSunSpec.eOperatingStateInverter := E_Symo_PV_OperatingState.eFaults;
				ELSIF 	arrBuffer_FC3[108] = 8 THEN stDataSunSpec.eOperatingStateInverter := E_Symo_PV_OperatingState.eStandby;
				ELSE 								stDataSunSpec.eOperatingStateInverter := E_Symo_PV_OperatingState.eNoDataReceived;
			END_IF
			//Next Step
			IF iStateModbus = 1 THEN
				fbMBRead_FC3.bExecute := FALSE;
				timDelay.IN := FALSE;
				iStateModbus := 2;
				stDataSunSpec.bError := FALSE; 
				stDataSunSpec.eErrorState := E_Symo_PV_Error.eNoError;
			END_IF
		END_IF
			
		//Error from Inverter
		IF NOT fbMBRead_FC3.bBusy AND NOT fbMBRead_FC3.bError AND timDelay.Q AND stDataSunSpec.eOperatingStateInverter = E_SunSpec_PV_OperatingState.eFaults THEN
			iStateModbus := 300;
			stDataSunSpec.eErrorState := E_Symo_PV_Error.eSymo10Error;
		END_IF
	 
		//Error or Timeout
		IF FPError_FC_3.Q OR timTimeout.Q THEN
			iStateModbus := 300;
			stDataSunSpec.eErrorState := E_SunSpec_PV_Error.eModbusTCPError;
		END_IF

	2://Wait and back to 1 step
		iStateModbus_CP := iStateModbus;
		
		iStateModbus := 1;
				
	300://Error
		iStateModbus_CP := iStateModbus;
		timDelay.IN := FALSE;
		fbMBRead_FC3.bExecute := FALSE;
		stDataSunSpec.bError := TRUE;
		iStateModbus := 1;							
END_CASE

(*------------------------------------------------------------------------------------------Modbus TCP Function---------------------------------------------------------------------------------------------*)

fbMBRead_FC3(	sIPAddr:= sIPAdress, 
				nTCPPort:= 502, 
				cbLength:= SIZEOF(arrBuffer_FC3), 
				pDestAddr:= ADR(arrBuffer_FC3), 
				tTimeout:= T#10S );

FPError_FC_3(CLK:= fbMBRead_FC3.bError, Q=> );

(*----------------------------------------------------------------------------------------Electric Meter Data----------------------------------------------------------------------------------------------*)

//Error and Warning
IF timDissableFunctions.Q THEN 
	fbElMeter.bWarning := TRUE; 
	fbElMeter.iWarningCode := 0; 
ELSE 
	fbElMeter.bWarning := FALSE; 
END_IF   

IF stDataSunSpec.bError OR Lynus_Standards.GVL_Energy.stNumberOfDevices.diNumberOfElectricMeters > Constants_Energy.diMaxNumberOfElectricMeters THEN 
	fbElMeter.bError := TRUE; 
ELSE 
	fbElMeter.bError := FALSE; 
END_IF  

IF Lynus_Standards.GVL_Energy.stNumberOfDevices.diNumberOfElectricMeters > Constants_Energy.diMaxNumberOfElectricMeters THEN 
	fbElMeter.iErrorCode := 1;
ELSIF stDataSunSpec.bError THEN 
	fbElMeter.iErrorCode := 0;
END_IF  

//Read Out Data done for EM Function
IF iStateModbus <> 2 THEN 
	fbElMeter.bReadOutDataDone := TRUE; 
ELSE 
	fbElMeter.bReadOutDataDone := FALSE; 
END_IF

//Function block for meter data
fbElMeter(
	bEnable:= bEnable AND NOT timDissableFunctions.Q, 
	bError:= , 
	bEnableReadOutFunction:= FALSE, 
	bWriteWithDelay:= TRUE,
	bPowerDataInvers:= TRUE, 
	bReadOutDataDone:= ,
	iTimeReadOutInterval:= , 
	iErrorCode:= , 
	iWarningCode:= , 
	lrTotalCounterEnergy_Consumption:= 0, 
	lrTotalCounterEnergy_Production:= , 
	lrCounterEnergyT1_Consumption:= 0, 
	lrCounterEnergyT2_Consumption:= 0, 
	lrCounterEnergyT1_Production:= , 
	lrCounterEnergyT2_Production:= 0, 
	lrCurrentL1:= , 
	lrVoltageL1N:= , 
	lrVoltageL1L2:= , 
	lrPowerL1:= 0, 
	lrCurrentL2:= , 
	lrVoltageL2N:= , 
	lrVoltageL2L3:= , 
	lrPowerL2:= 0, 
	lrCurrentL3:= , 
	lrVoltageL3N:= , 
	lrVoltageL3L1:= , 
	lrPowerL3:= 0, 
	lrPowerTotal:= , 
	lrFrequency:= , 
	lrReactivePowerTotal:= , 
	lrApparentPowerTotal:= , 
	tTimDelayOutput:= T#5S, 
	stDataEMOutPower=> , 
	stDataEMOutPowerDelay=> stDataEMPower_PV, 
	stDataEMOutCounter=> ,
	stDataEMOutCounterDelay=> stDataEMCounter_PV, 
	bReadOutMeter=> );
stDataSunSpec.lrPowerAcInverter := stDataEMPower_PV.lrPowerTotal;
(*-----------------------------------------------------------Handle data to Global structure for the Electric Meter system-----------------------------------------------------------------*)

CASE iStateGVLData OF
	
	0://Init Step
		byWaitInStep := 0;
		diCounterForGVL := 1;
	
	1://Wait for 4 Steps before clean al Data on GVL
		byWaitInStep := byWaitInStep + 1;
		IF byWaitInStep >= 4 AND fbNumberDevice.bNumberIsCalculatet THEN 
			iStateGVLData := 2; 
		END_IF
		//To much Devices, back to the Init step
		IF byWaitInStep >= 4 AND NOT fbNumberDevice.bNumberIsCalculatet THEN 
			iStateGVLData := 0; 
		END_IF	
			
	2://Clear all Data in GVL
		Lynus_Standards.GVL_Energy.stDataElectricMeters[diCounterForGVL].bEnabled := FALSE;	
		Lynus_Standards.GVL_Energy.stDataElectricMeters[diCounterForGVL].byErrorWarning := 0;
		Lynus_Standards.GVL_Energy.stDataElectricMeters[diCounterForGVL].lrCounterEnergyT1_Consumption := 0;
		Lynus_Standards.GVL_Energy.stDataElectricMeters[diCounterForGVL].lrCounterEnergyT1_Production := 0;
		Lynus_Standards.GVL_Energy.stDataElectricMeters[diCounterForGVL].lrCounterEnergyT2_Consumption := 0;
		Lynus_Standards.GVL_Energy.stDataElectricMeters[diCounterForGVL].lrCounterEnergyT2_Production := 0;
		Lynus_Standards.GVL_Energy.stDataElectricMeters[diCounterForGVL].lrPower := 0;
		Lynus_Standards.GVL_Energy.stDataElectricMeters[diCounterForGVL].lrPowerConsumption := 0;
		Lynus_Standards.GVL_Energy.stDataElectricMeters[diCounterForGVL].lrPowerConsumption := 0;
		Lynus_Standards.GVL_Energy.stDataElectricMeters[diCounterForGVL].lrPowerProduction := 0;
		Lynus_Standards.GVL_Energy.stDataElectricMeters[diCounterForGVL].lrTotalCounterEnergy_Consumption := 0;
		Lynus_Standards.GVL_Energy.stDataElectricMeters[diCounterForGVL].lrTotalCounterEnergy_Production := 0;
		
		diCounterForGVL := diCounterForGVL + 1;
		diCounterForGVL := LIMIT(0,diCounterForGVL,Constants_Energy.diMaxNumberOfElectricMeters);
		//Back to the init step
		IF diCounterForGVL >= Constants_Energy.diMaxNumberOfElectricMeters THEN 
			iStateGVLData := 0; 
		END_IF
END_CASE 	 

IF diNrOfEM_OUT_PV > 0 AND fbNumberDevice.bNumberIsCalculatet THEN
	Lynus_Standards.GVL_Energy.stDataElectricMeters[diNrOfEM_OUT_PV].bEnabled := fbElMeter.stDataEMOutPower.bEnabled;
	Lynus_Standards.GVL_Energy.stDataElectricMeters[diNrOfEM_OUT_PV].byErrorWarning := fbElMeter.stDataEMOutPower.byErrorWarning;
	Lynus_Standards.GVL_Energy.stDataElectricMeters[diNrOfEM_OUT_PV].lrCounterEnergyT1_Consumption := fbElMeter.stDataEMOutCounter.lrCounterEnergyT1_Consumption;
	Lynus_Standards.GVL_Energy.stDataElectricMeters[diNrOfEM_OUT_PV].lrCounterEnergyT1_Production := fbElMeter.stDataEMOutCounter.lrCounterEnergyT1_Production;
	Lynus_Standards.GVL_Energy.stDataElectricMeters[diNrOfEM_OUT_PV].lrCounterEnergyT2_Consumption := fbElMeter.stDataEMOutCounter.lrCounterEnergyT2_Consumption;
	Lynus_Standards.GVL_Energy.stDataElectricMeters[diNrOfEM_OUT_PV].lrCounterEnergyT2_Production := fbElMeter.stDataEMOutCounter.lrCounterEnergyT2_Production;		
	Lynus_Standards.GVL_Energy.stDataElectricMeters[diNrOfEM_OUT_PV].lrPower := fbElMeter.stDataEMOutPower.lrPowerTotal;
	Lynus_Standards.GVL_Energy.stDataElectricMeters[diNrOfEM_OUT_PV].lrPowerConsumption := fbElMeter.stDataEMOutPower.lrPowerConsumption;
	Lynus_Standards.GVL_Energy.stDataElectricMeters[diNrOfEM_OUT_PV].lrPowerProduction := fbElMeter.stDataEMOutPower.lrPowerProduction;
	Lynus_Standards.GVL_Energy.stDataElectricMeters[diNrOfEM_OUT_PV].lrTotalCounterEnergy_Consumption := fbElMeter.stDataEMOutCounter.lrTotalCounterEnergy_Consumption;
	Lynus_Standards.GVL_Energy.stDataElectricMeters[diNrOfEM_OUT_PV].lrTotalCounterEnergy_Production := fbElMeter.stDataEMOutCounter.lrTotalCounterEnergy_Production;
END_IF

(*----------------------------------------------------------Save persistent data----------------------------------------------------------------*)

arrPD[1](lrValue:= BOOL_TO_LREAL(bEnable), bEventBasedActive=> );
arrPD[2](lrValue:= BYTE_TO_LREAL(byUnitID_Inverter), bEventBasedActive=> );
PD_String(sText:= sIPAdress, bEventBasedActive=> );

END_FUNCTION_BLOCK

// ---- FBs/Soltop/M_Tec/FB_HP_Soltop_M_Tec_Modular.TcPOU
FUNCTION_BLOCK FB_HP_Soltop_M_Tec_Modular
VAR_INPUT PERSISTENT
	bEnable									: BOOL;												//{#lynus.ag#()} //Enable the Fuctionblock and his logic
	bPowerDataInvers						: BOOL;												//With True its possible to invert all received power data from the electric meter
	byUnitID								: BYTE;												//Unit ID fromt the Soltop M-Tec Modbus Server(0 to 255)
	diNrOfEMS_IN							: DINT;												//Number of EMS what control this Device.
	diNrOfEM_IN_HP							: DINT;												//Number of the electric meter for incoming power data. (Power Data for this Device)
	sIPAdress								: STRING(15);										//IP Adress from the oltop M-Tec Modbus Server
	stSetupHP								: ST_Setup_HP;										//{#lynus.ag#()} //Setup heating pump
END_VAR
VAR_INPUT
END_VAR
VAR_OUTPUT
	stDataHP								: ST_HP_Output;										//{#lynus.ag#()} //Output Data Heating pump
	stDataTempS								: ST_Temperature_Output;							//Temperature output data
	diNrOfHP_OUT							: DINT;												//Active Number from the heating pump for using on other functions		
	diNrOfTempS_OUT_ServiceWaterTop			: DINT;												//Active Number from the Temperature Sensor for using on other functions
END_VAR
VAR
	{attribute 'hide'}
	fbHP									: FB_HeatingPump;									//Function block for heating pump
	{attribute 'hide'}
	fbNumberDevice							: FB_NumberOfDevice;								//Function block to calcualte the number of the Device
	{attribute 'hide'}
	fbNumberDevice_Temp						: FB_NumberOfDevice;								//Function block to calcualte the number of the Device
	{attribute 'hide'}
	fbTempS									: FB_TempSensor_M50_P200;							//Function for Temperature Sensor
	fbDIExternalLock						: FB_XL1XXX_DI;										//Digital Input from external loock signal
	{attribute 'hide'}
	timDissableFunctions					: TON;												//Timer to dissable the Function after Lynus_Standards.Constants_General.tTimeDissableLynusFunctions Days without connection to the Lynus Cloud
	{attribute 'hide'}
	timResetConnectionOnGVL					: TON;												//Timer to try reset the connection Flag on the GVL. (When somebody delete the Connection Function and make only a onlinechange)
	{attribute 'hide'}
	timGetTime								: TON;												//Timer to activate the function tho read out the windows system time
	{attribute 'hide'}
	timDelay								: TON;												//Timer for Delay between Requests
	{attribute 'hide'}
	timTimeout								: TON;												//Timer for Timeout
	{attribute 'hide'}
	timSurplusForTemp						: TON;												//Timer to set the Temperature in the whater boiler after this delay on a higher value
	{attribute 'hide'}
	FNReset									: F_TRIG;											//Internal negative edge
	{attribute 'hide'}
	FPEnable								: R_TRIG;											//Internal positive Edge
	{attribute 'hide'}
	FNTimDissable							: F_TRIG;											//Internal negative Edge
	{attribute 'hide'}
	FPError_FC_3							: R_TRIG;											//Internal positive Edge
	{attribute 'hide'}
	FPError_FC_6							: R_TRIG;											//Internal positive Edge
	{attribute 'hide'}
	fbGetSystemTime							: NT_GetTime;										//Function to read out the windows system time on the local plc
	{attribute 'hide'}
	arrPD									: ARRAY[1..21] OF FB_PersistentData_Number;			//Function to save persistent data
	{attribute 'hide'}
	fbPDString								: FB_PersistentData_String;							//Function to save persistent string data
	{attribute 'hide'}
	fbMBRead_FC3							: FB_MBReadRegs;									//Modbus Read Function (FC3)
	{attribute 'hide'}
	fbMBWrite_FC6							: FB_MBWriteSingleReg;								//Modbus Write Function (FC6)
	{attribute 'hide'}
	arrCounterForGVL						: ARRAY[1..2] OF DINT;								//Counter to clean old data on GVL
	{attribute 'hide'}
	arrBuffer_FC3							: ARRAY[1..8] OF WORD;								//Buffer with Data from FC3
	{attribute 'hide'}
	bGroupErrorHP							: BOOL;												//Group Error from the Heating Pump
	{attribute 'hide'}
	bHPIsRunning							: BOOL;												//Feedback from the HP if its running or not
	{attribute 'hide'}
	bErrorTempSensorBoilerServiceWaterTop	: BOOL;												//Error for the Temp Senor top in the service water boiler
	{attribute 'hide'}
	bMBTCPError								: BOOL;												//Modbus TCP Error
	{attribute 'hide'}
	byWaitInStep							: BYTE;												//Wait in Step before start to clean data on PLC
	{attribute 'hide'}
	iStateGVLData							: INT;												//State machine to handle the data on the GVL
	{attribute 'hide'}
	iStateModbusRead						: INT;												//State variable for Statemachine
	{attribute 'hide'}
	iStateModbusWrite						: INT;												//State variable for Statemachine
	{attribute 'hide'}
	iStateModbusError						: INT;												//State variable for Statemachine
	{attribute 'hide'}
	iStateModbus_CP							: INT;												//Compare State variable
	{attribute 'hide'}
	diNumberOfActiveBatterys				: DINT;												//Number of active batterys
	{attribute 'hide'}
	diNumberOfBatteryInverterInEPO			: DINT;												//Number of battery inverters that work in Emergency Power operation 
	{attribute 'hide'}
	diLPForGVL								: DINT;												//Loop to clean old data on GVL
	{attribute 'hide'}	
	dwSumSOC								: DWORD;											//Sum of the SOC from all batterys
	{attribute 'hide'}
	rNewPowerToHP							: REAL;												//New surplus power fpr the HP in W
	{attribute 'hide'}
	lrGridPower								: LREAL;											//Grid power in kW
	{attribute 'hide'}
	lrSizeGridConnection					: LREAL;											//Size of the complete grid connection
	{attribute 'hide'}
	liLPBatteryData							: LINT;												//Loop to check some data from batterys
	{attribute 'hide'}
	liLPInEPO								: LINT;												//Loop to check if 1 or more battery inverters build a island grid	
	{attribute 'hide'}
	liLPGridData							: LINT;												//Loop to check some grid data
END_VAR
VAR PERSISTENT
	{attribute 'conditionalshow'}
	diNrOfEMS_IN_CP							: DINT;												//Number of EMS what control this Device to compare with the original
END_VAR

//Creator : Kai Ebensperger
//Company : Lynus AG
//Date : 12.08.2021
//Version : 1.0.0.0

//With this function block its possible to control a Heating pump from the Factory Soltop
//The communication is over Modbus TCP.
//The Device on the Soltop side is called M-Tec Modbus Server.
//The excess power can be transferred to this pump linearly as it is modulating. The power can be transferred in watts.
//Versions that are supported : 20210531
//This function work only with the Headpump what is in the documentation under [0]

//NOTE for diNr.....Designation => 
//_IN = Here Data come in from other Functions or go out to other functions about the GVL
//_OUT = Here Data go out to other functions about the GVL

(*------------------------------------------------------------Limits----------------------------------------------------------------------------------*)

